LIN {X 0,Y 199.376,Z 843.056,A -85,B 0,C 180,E1 -21344.287,E2 -21344.287} C_VEL
LIN {X 0,Y 201.471,Z 836.822,A -85,B 0,C 180,E1 -21347.773,E2 -21347.773} C_VEL
LIN {X 0,Y 203.749,Z 830.038,A -85,B 0,C 180,E1 -21350.701,E2 -21350.701} C_VEL
LIN {X 0,Y 206.319,Z 821.68,A -85,B 0,C 180,E1 -21353.542,E2 -21353.542} C_VEL
LIN {X 0,Y 208.991,Z 812.769,A -85,B 0,C 180,E1 -21355.925,E2 -21355.925} C_VEL
LIN {X 0,Y 212.11,Z 801.995,A -85,B 0,C 180,E1 -21358.176,E2 -21358.176} C_VEL
LIN {X 0,Y 214.813,Z 791.098,A -85,B 0,C 180,E1 -21359.931,E2 -21359.931} C_VEL
LIN {X 0,Y 217.315,Z 778.908,A -85,B 0,C 180,E1 -21361.433,E2 -21361.433} C_VEL
LIN {X 0,Y 219.233,Z 767.366,A -85,B 0,C 180,E1 -21362.478,E2 -21362.478} C_VEL
LIN {X 0,Y 220.897,Z 754.07,A -85,B 0,C 180,E1 -21363.276,E2 -21363.276} C_VEL
LIN {X 0,Y 221.812,Z 738.89,A -85,B 0,C 180,E1 -21363.832,E2 -21363.832} C_VEL
LIN {X 0,Y 223.844,Z 690.241,A -85,B 0,C 180,E1 -21365.33,E2 -21365.33} C_VEL
LIN {X 0,Y 221.912,Z 665.137,A -85,B 0,C 180,E1 -21366.665,E2 -21366.665} C_VEL
LIN {X 0,Y 218.953,Z 639.437,A -85,B 0,C 180,E1 -21368.282,E2 -21368.282} C_VEL
LIN {X 0,Y 218.22,Z 633.043,A -85,B 0,C 180,E1 -21368.759,E2 -21368.759} C_VEL
LIN {X 0,Y 218.577,Z 624.565,A -85,B 0,C 180,E1 -21370.022,E2 -21370.022} C_VEL
LIN {X 0,Y 214.349,Z 607.039,A -85,B 0,C 180,E1 -21373.836,E2 -21373.836} C_VEL
LIN {X 0,Y 212.098,Z 598.465,A -85,B 0,C 180,E1 -21375.905,E2 -21375.905} C_VEL
LIN {X 0,Y 207.217,Z 589.004,A -85,B 0,C 180,E1 -21379.24,E2 -21379.24} C_VEL
LIN {X 0,Y 203.836,Z 583.546,A -85,B 0,C 180,E1 -21381.639,E2 -21381.639} C_VEL
LIN {X 0,Y 201.926,Z 579.961,A -85,B 0,C 180,E1 -21383.181,E2 -21383.181} C_VEL
LIN {X 0,Y 200.29,Z 577.767,A -85,B 0,C 180,E1 -21384.366,E2 -21384.366} C_VEL
LIN {X 0,Y 199.63,Z 575.61,A -85,B 0,C 180,E1 -21385.255,E2 -21385.255} C_VEL
LIN {X 0,Y 199.697,Z 575.587,A -85,B 0,C 180,E1 -21388.136,E2 -21388.136} C_VEL
LIN {X 0,Y 199.69,Z 575.605,A -85,B 0,C 180,E1 -21392.772,E2 -21392.772} C_VEL
LIN {X 0,Y 199.718,Z 575.592,A -85,B 0,C 180,E1 -21397.227,E2 -21397.227} C_VEL
LIN {X 0,Y 199.799,Z 575.564,A -85,B 0,C 180,E1 -21401.759,E2 -21401.759} C_VEL
LIN {X 0,Y 199.837,Z 575.594,A -85,B 0,C 180,E1 -21405.748,E2 -21405.748} C_VEL
LIN {X 0,Y 200.026,Z 575.533,A -85,B 0,C 180,E1 -21409.882,E2 -21409.882} C_VEL
LIN {X 0,Y 200.026,Z 575.568,A -85,B 0,C 180,E1 -21413.949,E2 -21413.949} C_VEL
LIN {X 0,Y 200.323,Z 575.496,A -85,B 0,C 180,E1 -21417.99,E2 -21417.99} C_VEL
LIN {X 0,Y 200.479,Z 575.502,A -85,B 0,C 180,E1 -21420,E2 -21420} C_VEL
LIN {X 0,Y 200.03,Z 575.536,A -85,B 0,C 180,E1 -21424.03,E2 -21424.03} C_VEL
LIN {X 0,Y 200.114,Z 575.554,A -85,B 0,C 180,E1 -21428.076,E2 -21428.076} C_VEL
LIN {X 0,Y 200.04,Z 575.55,A -85,B 0,C 180,E1 -21430.347,E2 -21430.347} C_VEL
LIN {X 0,Y 199.808,Z 575.596,A -85,B 0,C 180,E1 -21436.343,E2 -21436.343} C_VEL
LIN {X 0,Y 199.704,Z 575.587,A -85,B 0,C 180,E1 -21440.605,E2 -21440.605} C_VEL
LIN {X 0,Y 199.676,Z 575.589,A -85,B 0,C 180,E1 -21444.984,E2 -21444.984} C_VEL
LIN {X 0,Y 199.66,Z 575.671,A -85,B 0,C 180,E1 -21449.597,E2 -21449.597} C_VEL
LIN {X 0,Y 200.238,Z 577.621,A -85,B 0,C 180,E1 -21450.592,E2 -21450.592} C_VEL
LIN {X 0,Y 201.666,Z 580.137,A -85,B 0,C 180,E1 -21452.107,E2 -21452.107} C_VEL
LIN {X 0,Y 204.816,Z 586.849,A -85,B 0,C 180,E1 -21455.686,E2 -21455.686} C_VEL
LIN {X 0,Y 208.857,Z 596.996,A -85,B 0,C 180,E1 -21460.373,E2 -21460.373} C_VEL
LIN {X 0,Y 212.009,Z 606.282,A -85,B 0,C 180,E1 -21464.119,E2 -21464.119} C_VEL
LIN {X 0,Y 214.73,Z 615.526,A -85,B 0,C 180,E1 -21467.426,E2 -21467.426} C_VEL
LIN {X 0,Y 217.067,Z 625.231,A -85,B 0,C 180,E1 -21470.547,E2 -21470.547} C_VEL
LIN {X 0,Y 217.574,Z 627.419,A -85,B 0,C 180,E1 -21471.118,E2 -21471.118} C_VEL
LIN {X 0,Y 221.203,Z 635.829,A -85,B 0,C 180,E1 -21472.215,E2 -21472.215} C_VEL
LIN {X 0,Y 225.045,Z 664.563,A -85,B 0,C 180,E1 -21474.094,E2 -21474.094} C_VEL
LIN {X 0,Y 225.417,Z 668.676,A -85,B 0,C 180,E1 -21474.321,E2 -21474.321} C_VEL
LIN {X 0,Y 222.027,Z 739.582,A -85,B 0,C 180,E1 -21476.497,E2 -21476.497} C_VEL
LIN {X 0,Y 220.853,Z 752.225,A -85,B 0,C 180,E1 -21477.181,E2 -21477.181} C_VEL
LIN {X 0,Y 219.127,Z 764.44,A -85,B 0,C 180,E1 -21478.183,E2 -21478.183} C_VEL
LIN {X 0,Y 217.191,Z 775.07,A -85,B 0,C 180,E1 -21479.358,E2 -21479.358} C_VEL
LIN {X 0,Y 214.454,Z 787.114,A -85,B 0,C 180,E1 -21481.092,E2 -21481.092} C_VEL
LIN {X 0,Y 211.658,Z 797.714,A -85,B 0,C 180,E1 -21483.1,E2 -21483.1} C_VEL
LIN {X 0,Y 208.872,Z 807.539,A -85,B 0,C 180,E1 -21485.485,E2 -21485.485} C_VEL
LIN {X 0,Y 206.3,Z 815.759,A -85,B 0,C 180,E1 -21487.991,E2 -21487.991} C_VEL
LIN {X 0,Y 203.644,Z 823.224,A -85,B 0,C 180,E1 -21490.86,E2 -21490.86} C_VEL
LIN {X 0,Y 201.56,Z 829.214,A -85,B 0,C 180,E1 -21493.801,E2 -21493.801} C_VEL
LIN {X 0,Y 199.915,Z 833.946,A -85,B 0,C 180,E1 -21496.789,E2 -21496.789} C_VEL
LIN {X 0,Y 198.731,Z 837.559,A -85,B 0,C 180,E1 -21499.814,E2 -21499.814} C_VEL
LIN {X 0,Y 198.161,Z 839.419,A -85,B 0,C 180,E1 -21501.843,E2 -21501.843} C_VEL
LIN {X 0,Y 197.641,Z 841.261,A -85,B 0,C 180,E1 -21504.667,E2 -21504.667} C_VEL
LIN {X 0,Y 197.397,Z 842.439,A -85,B 0,C 180,E1 -21507.958,E2 -21507.958} C_VEL
LIN {X 0,Y 197.399,Z 842.669,A -85,B 0,C 180,E1 -21509.998,E2 -21509.998} C_VEL
LIN {X 0,Y 197.379,Z 842.473,A -85,B 0,C 180,E1 -21512.039,E2 -21512.039} C_VEL
LIN {X 0,Y 197.765,Z 840.915,A -85,B 0,C 180,E1 -21516.118,E2 -21516.118} C_VEL
LIN {X 0,Y 198.157,Z 839.543,A -85,B 0,C 180,E1 -21518.154,E2 -21518.154} C_VEL
LIN {X 0,Y 199.041,Z 836.661,A -85,B 0,C 180,E1 -21521.196,E2 -21521.196} C_VEL
LIN {X 0,Y 200.358,Z 832.739,A -85,B 0,C 180,E1 -21524.212,E2 -21524.212} C_VEL
LIN {X 0,Y 202.134,Z 827.658,A -85,B 0,C 180,E1 -21527.188,E2 -21527.188} C_VEL
LIN {X 0,Y 204.412,Z 821.25,A -85,B 0,C 180,E1 -21530.107,E2 -21530.107} C_VEL
LIN {X 0,Y 207.218,Z 813.27,A -85,B 0,C 180,E1 -21532.954,E2 -21532.954} C_VEL
LIN {X 0,Y 209.758,Z 804.815,A -85,B 0,C 180,E1 -21535.376,E2 -21535.376} C_VEL
LIN {X 0,Y 212.511,Z 795.054,A -85,B 0,C 180,E1 -21537.578,E2 -21537.578} C_VEL
LIN {X 0,Y 215.082,Z 785.125,A -85,B 0,C 180,E1 -21539.347,E2 -21539.347} C_VEL
LIN {X 0,Y 217.429,Z 774.318,A -85,B 0,C 180,E1 -21540.87,E2 -21540.87} C_VEL
LIN {X 0,Y 219.557,Z 762.357,A -85,B 0,C 180,E1 -21542.149,E2 -21542.149} C_VEL
LIN {X 0,Y 221.179,Z 749.901,A -85,B 0,C 180,E1 -21543.1,E2 -21543.1} C_VEL
LIN {X 0,Y 222.278,Z 737.222,A -85,B 0,C 180,E1 -21543.728,E2 -21543.728} C_VEL
LIN {X 0,Y 225.333,Z 671.392,A -85,B 0,C 180,E1 -21545.738,E2 -21545.738} C_VEL
LIN {X 0,Y 223.232,Z 655.911,A -85,B 0,C 180,E1 -21546.737,E2 -21546.737} C_VEL
LIN {X 0,Y 219.777,Z 634.786,A -85,B 0,C 180,E1 -21548.273,E2 -21548.273} C_VEL
LIN {X 0,Y 216.645,Z 627.6,A -85,B 0,C 180,E1 -21549.285,E2 -21549.285} C_VEL
LIN {X 0,Y 215.672,Z 627.608,A -85,B 0,C 180,E1 -21549.503,E2 -21549.503} C_VEL
LIN {X 0,Y 214.082,Z 629.763,A -85,B 0,C 180,E1 -21549.702,E2 -21549.702} C_VEL
LIN {X 0,Y 212.932,Z 631.087,A -85,B 0,C 180,E1 -21549.903,E2 -21549.903} C_VEL
LIN {X 0,Y 211.461,Z 631.109,A -85,B 0,C 180,E1 -21550.237,E2 -21550.237} C_VEL
LIN {X 0,Y 210.574,Z 629.639,A -85,B 0,C 180,E1 -21550.506,E2 -21550.506} C_VEL
LIN {X 0,Y 210.223,Z 628.001,A -85,B 0,C 180,E1 -21550.671,E2 -21550.671} C_VEL
LIN {X 0,Y 209.975,Z 627.554,A -85,B 0,C 180,E1 -21550.868,E2 -21550.868} C_VEL
LIN {X 0,Y 209.013,Z 661.135,A -85,B 0,C 180,E1 -21552.558,E2 -21552.558} C_VEL
LIN {X 0,Y 208.249,Z 675.161,A -85,B 0,C 180,E1 -21553.658,E2 -21553.658} C_VEL
LIN {X 0,Y 207.163,Z 689.066,A -85,B 0,C 180,E1 -21555.193,E2 -21555.193} C_VEL
LIN {X 0,Y 205.976,Z 701.306,A -85,B 0,C 180,E1 -21556.967,E2 -21556.967} C_VEL
LIN {X 0,Y 204.576,Z 713.727,A -85,B 0,C 180,E1 -21559.252,E2 -21559.252} C_VEL
LIN {X 0,Y 203.312,Z 723.628,A -85,B 0,C 180,E1 -21561.521,E2 -21561.521} C_VEL
LIN {X 0,Y 202.091,Z 733.699,A -85,B 0,C 180,E1 -21564.373,E2 -21564.373} C_VEL
LIN {X 0,Y 201.177,Z 741.175,A -85,B 0,C 180,E1 -21566.97,E2 -21566.97} C_VEL
LIN {X 0,Y 200.519,Z 748.385,A -85,B 0,C 180,E1 -21570.036,E2 -21570.036} C_VEL
LIN {X 0,Y 200.122,Z 753.722,A -85,B 0,C 180,E1 -21572.836,E2 -21572.836} C_VEL
LIN {X 0,Y 200.06,Z 758.466,A -85,B 0,C 180,E1 -21575.969,E2 -21575.969} C_VEL
LIN {X 0,Y 200.524,Z 762.436,A -85,B 0,C 180,E1 -21579.483,E2 -21579.483} C_VEL
LIN {X 0,Y 201.076,Z 764.264,A -85,B 0,C 180,E1 -21581.665,E2 -21581.665} C_VEL
LIN {X 0,Y 201.845,Z 765.542,A -85,B 0,C 180,E1 -21583.826,E2 -21583.826} C_VEL
LIN {X 0,Y 202.818,Z 766.369,A -85,B 0,C 180,E1 -21585.978,E2 -21585.978} C_VEL
LIN {X 0,Y 204.018,Z 766.722,A -85,B 0,C 180,E1 -21588.072,E2 -21588.072} C_VEL
LIN {X 0,Y 206.228,Z 766.345,A -85,B 0,C 180,E1 -21591.204,E2 -21591.204} C_VEL
LIN {X 0,Y 208.844,Z 764.942,A -85,B 0,C 180,E1 -21594.206,E2 -21594.206} C_VEL
LIN {X 0,Y 211.219,Z 763.1,A -85,B 0,C 180,E1 -21596.524,E2 -21596.524} C_VEL
LIN {X 0,Y 214.247,Z 760.206,A -85,B 0,C 180,E1 -21599.06,E2 -21599.06} C_VEL
LIN {X 0,Y 218.012,Z 755.835,A -85,B 0,C 180,E1 -21601.847,E2 -21601.847} C_VEL
LIN {X 0,Y 222.275,Z 750.161,A -85,B 0,C 180,E1 -21604.534,E2 -21604.534} C_VEL
LIN {X 0,Y 226.866,Z 742.967,A -85,B 0,C 180,E1 -21607.118,E2 -21607.118} C_VEL
LIN {X 0,Y 231.669,Z 734.065,A -85,B 0,C 180,E1 -21609.605,E2 -21609.605} C_VEL
LIN {X 0,Y 236.461,Z 723.753,A -85,B 0,C 180,E1 -21611.791,E2 -21611.791} C_VEL
LIN {X 0,Y 240.467,Z 713.449,A -85,B 0,C 180,E1 -21613.522,E2 -21613.522} C_VEL
LIN {X 0,Y 244.029,Z 701.968,A -85,B 0,C 180,E1 -21615.038,E2 -21615.038} C_VEL
LIN {X 0,Y 245.05,Z 696.962,A -85,B 0,C 180,E1 -21615.739,E2 -21615.739} C_VEL
LIN {X 0,Y 245.616,Z 689.046,A -85,B 0,C 180,E1 -21617.134,E2 -21617.134} C_VEL
LIN {X 0,Y 245.924,Z 680.855,A -85,B 0,C 180,E1 -21618.409,E2 -21618.409} C_VEL
LIN {X 0,Y 246.461,Z 675.44,A -85,B 0,C 180,E1 -21618.918,E2 -21618.918} C_VEL
LIN {X 0,Y 249.571,Z 650.857,A -85,B 0,C 180,E1 -21620.206,E2 -21620.206} C_VEL
LIN {X 0,Y 250.153,Z 646.426,A -85,B 0,C 180,E1 -21620.424,E2 -21620.424} C_VEL
LIN {X 0,Y 248.082,Z 641.857,A -85,B 0,C 180,E1 -21622.351,E2 -21622.351} C_VEL
LIN {X 0,Y 246.401,Z 638.478,A -85,B 0,C 180,E1 -21624.264,E2 -21624.264} C_VEL
LIN {X 0,Y 244.337,Z 636.415,A -85,B 0,C 180,E1 -21626.921,E2 -21626.921} C_VEL
LIN {X 0,Y 242.313,Z 636.359,A -85,B 0,C 180,E1 -21631.471,E2 -21631.471} C_VEL
LIN {X 0,Y 242.029,Z 637.453,A -85,B 0,C 180,E1 -21633.593,E2 -21633.593} C_VEL
LIN {X 0,Y 242.252,Z 640.017,A -85,B 0,C 180,E1 -21636.149,E2 -21636.149} C_VEL
LIN {X 0,Y 243.693,Z 646.744,A -85,B 0,C 180,E1 -21640.038,E2 -21640.038} C_VEL
LIN {X 0,Y 244.457,Z 650.053,A -85,B 0,C 180,E1 -21641.394,E2 -21641.394} C_VEL
LIN {X 0,Y 245.563,Z 654.466,A -85,B 0,C 180,E1 -21642.967,E2 -21642.967} C_VEL
LIN {X 0,Y 246.515,Z 658.782,A -85,B 0,C 180,E1 -21644.224,E2 -21644.224} C_VEL
LIN {X 0,Y 245.896,Z 673.924,A -85,B 0,C 180,E1 -21645.758,E2 -21645.758} C_VEL
LIN {X 0,Y 244.774,Z 689.882,A -85,B 0,C 180,E1 -21646.984,E2 -21646.984} C_VEL
LIN {X 0,Y 244.081,Z 696.611,A -85,B 0,C 180,E1 -21647.382,E2 -21647.382} C_VEL
LIN {X 0,Y 241.31,Z 711.484,A -85,B 0,C 180,E1 -21648.087,E2 -21648.087} C_VEL
LIN {X 0,Y 237.61,Z 725.575,A -85,B 0,C 180,E1 -21648.987,E2 -21648.987} C_VEL
LIN {X 0,Y 233.041,Z 739.08,A -85,B 0,C 180,E1 -21650.147,E2 -21650.147} C_VEL
LIN {X 0,Y 227.776,Z 751.778,A -85,B 0,C 180,E1 -21651.617,E2 -21651.617} C_VEL
LIN {X 0,Y 222.272,Z 763.259,A -85,B 0,C 180,E1 -21653.361,E2 -21653.361} C_VEL
LIN {X 0,Y 216.595,Z 773.724,A -85,B 0,C 180,E1 -21655.403,E2 -21655.403} C_VEL
LIN {X 0,Y 210.95,Z 783.143,A -85,B 0,C 180,E1 -21657.79,E2 -21657.79} C_VEL
LIN {X 0,Y 210.163,Z 784.755,A -85,B 0,C 180,E1 -21658.22,E2 -21658.22} C_VEL
LIN {X 0,Y 207.263,Z 796.997,A -85,B 0,C 180,E1 -21659.992,E2 -21659.992} C_VEL
LIN {X 0,Y 204.247,Z 807.724,A -85,B 0,C 180,E1 -21662.044,E2 -21662.044} C_VEL
LIN {X 0,Y 200.959,Z 818.25,A -85,B 0,C 180,E1 -21664.636,E2 -21664.636} C_VEL
LIN {X 0,Y 198.092,Z 827.068,A -85,B 0,C 180,E1 -21667.467,E2 -21667.467} C_VEL
LIN {X 0,Y 195.445,Z 834.658,A -85,B 0,C 180,E1 -21670.574,E2 -21670.574} C_VEL
LIN {X 0,Y 193.663,Z 839.604,A -85,B 0,C 180,E1 -21673.125,E2 -21673.125} C_VEL
LIN {X 0,Y 192.069,Z 844.394,A -85,B 0,C 180,E1 -21676.243,E2 -21676.243} C_VEL
LIN {X 0,Y 191.044,Z 848.058,A -85,B 0,C 180,E1 -21679.403,E2 -21679.403} C_VEL
LIN {X 0,Y 190.578,Z 849.948,A -85,B 0,C 180,E1 -21681.519,E2 -21681.519} C_VEL
LIN {X 0,Y 190.321,Z 851.372,A -85,B 0,C 180,E1 -21683.642,E2 -21683.642} C_VEL
LIN {X 0,Y 190.238,Z 852.44,A -85,B 0,C 180,E1 -21685.921,E2 -21685.921} C_VEL
LIN {X 0,Y 190.381,Z 853.216,A -85,B 0,C 180,E1 -21690.002,E2 -21690.002} C_VEL
LIN {X 0,Y 190.235,Z 852.424,A -85,B 0,C 180,E1 -21694.064,E2 -21694.064} C_VEL
LIN {X 0,Y 190.324,Z 851.34,A -85,B 0,C 180,E1 -21696.362,E2 -21696.362} C_VEL
LIN {X 0,Y 190.582,Z 849.898,A -85,B 0,C 180,E1 -21698.484,E2 -21698.484} C_VEL
LIN {X 0,Y 191.316,Z 846.911,A -85,B 0,C 180,E1 -21701.658,E2 -21701.658} C_VEL
LIN {X 0,Y 192.463,Z 842.862,A -85,B 0,C 180,E1 -21704.811,E2 -21704.811} C_VEL
LIN {X 0,Y 194.701,Z 836.629,A -85,B 0,C 180,E1 -21708.413,E2 -21708.413} C_VEL
LIN {X 0,Y 197.054,Z 829.98,A -85,B 0,C 180,E1 -21711.379,E2 -21711.379} C_VEL
LIN {X 0,Y 199.351,Z 822.889,A -85,B 0,C 180,E1 -21713.919,E2 -21713.919} C_VEL
LIN {X 0,Y 202.025,Z 814.508,A -85,B 0,C 180,E1 -21716.332,E2 -21716.332} C_VEL
LIN {X 0,Y 205.192,Z 804.136,A -85,B 0,C 180,E1 -21718.655,E2 -21718.655} C_VEL
LIN {X 0,Y 208.344,Z 792.457,A -85,B 0,C 180,E1 -21720.679,E2 -21720.679} C_VEL
LIN {X 0,Y 210.886,Z 780.679,A -85,B 0,C 180,E1 -21722.224,E2 -21722.224} C_VEL
LIN {X 0,Y 213.068,Z 768.472,A -85,B 0,C 180,E1 -21723.398,E2 -21723.398} C_VEL
LIN {X 0,Y 214.843,Z 755.964,A -85,B 0,C 180,E1 -21724.209,E2 -21724.209} C_VEL
LIN {X 0,Y 215.781,Z 742.593,A -85,B 0,C 180,E1 -21724.761,E2 -21724.761} C_VEL
LIN {X 0,Y 218.04,Z 690.784,A -85,B 0,C 180,E1 -21726.393,E2 -21726.393} C_VEL
LIN {X 0,Y 216.288,Z 666.684,A -85,B 0,C 180,E1 -21727.715,E2 -21727.715} C_VEL
LIN {X 0,Y 213.485,Z 641.41,A -85,B 0,C 180,E1 -21729.362,E2 -21729.362} C_VEL
LIN {X 0,Y 212.474,Z 633.523,A -85,B 0,C 180,E1 -21729.924,E2 -21729.924} C_VEL
LIN {X 0,Y 212.772,Z 627.098,A -85,B 0,C 180,E1 -21730.924,E2 -21730.924} C_VEL
LIN {X 0,Y 208.979,Z 610.361,A -85,B 0,C 180,E1 -21734.729,E2 -21734.729} C_VEL
LIN {X 0,Y 206.944,Z 602.434,A -85,B 0,C 180,E1 -21736.722,E2 -21736.722} C_VEL
LIN {X 0,Y 202.859,Z 594.437,A -85,B 0,C 180,E1 -21739.659,E2 -21739.659} C_VEL
LIN {X 0,Y 199.698,Z 589.173,A -85,B 0,C 180,E1 -21741.984,E2 -21741.984} C_VEL
LIN {X 0,Y 197.193,Z 584.939,A -85,B 0,C 180,E1 -21743.98,E2 -21743.98} C_VEL
LIN {X 0,Y 194.973,Z 580.965,A -85,B 0,C 180,E1 -21746.004,E2 -21746.004} C_VEL
LIN {X 0,Y 193.382,Z 578.923,A -85,B 0,C 180,E1 -21747.4,E2 -21747.4} C_VEL
LIN {X 0,Y 192.624,Z 576.465,A -85,B 0,C 180,E1 -21748.52,E2 -21748.52} C_VEL
LIN {X 0,Y 192.668,Z 576.484,A -85,B 0,C 180,E1 -21751.692,E2 -21751.692} C_VEL
LIN {X 0,Y 192.688,Z 576.457,A -85,B 0,C 180,E1 -21756.346,E2 -21756.346} C_VEL
LIN {X 0,Y 192.734,Z 576.445,A -85,B 0,C 180,E1 -21761.459,E2 -21761.459} C_VEL
LIN {X 0,Y 192.765,Z 576.471,A -85,B 0,C 180,E1 -21765.214,E2 -21765.214} C_VEL
LIN {X 0,Y 192.949,Z 576.413,A -85,B 0,C 180,E1 -21769.567,E2 -21769.567} C_VEL
LIN {X 0,Y 192.988,Z 576.446,A -85,B 0,C 180,E1 -21773.728,E2 -21773.728} C_VEL
LIN {X 0,Y 193.265,Z 576.374,A -85,B 0,C 180,E1 -21777.916,E2 -21777.916} C_VEL
LIN {X 0,Y 193.443,Z 576.377,A -85,B 0,C 180,E1 -21780,E2 -21780} C_VEL
LIN {X 0,Y 192.977,Z 576.412,A -85,B 0,C 180,E1 -21784.177,E2 -21784.177} C_VEL
LIN {X 0,Y 193.065,Z 576.435,A -85,B 0,C 180,E1 -21788.373,E2 -21788.373} C_VEL
LIN {X 0,Y 192.813,Z 576.434,A -85,B 0,C 180,E1 -21792.633,E2 -21792.633} C_VEL
LIN {X 0,Y 192.761,Z 576.463,A -85,B 0,C 180,E1 -21796.959,E2 -21796.959} C_VEL
LIN {X 0,Y 192.641,Z 576.476,A -85,B 0,C 180,E1 -21801.397,E2 -21801.397} C_VEL
LIN {X 0,Y 192.668,Z 576.465,A -85,B 0,C 180,E1 -21804.224,E2 -21804.224} C_VEL
LIN {X 0,Y 192.615,Z 576.495,A -85,B 0,C 180,E1 -21806.404,E2 -21806.404} C_VEL
LIN {X 0,Y 193.635,Z 579.261,A -85,B 0,C 180,E1 -21808.154,E2 -21808.154} C_VEL
LIN {X 0,Y 194.623,Z 580.578,A -85,B 0,C 180,E1 -21809.2,E2 -21809.2} C_VEL
LIN {X 0,Y 195.237,Z 582.498,A -85,B 0,C 180,E1 -21810.263,E2 -21810.263} C_VEL
LIN {X 0,Y 196.603,Z 585.04,A -85,B 0,C 180,E1 -21811.821,E2 -21811.821} C_VEL
LIN {X 0,Y 200.155,Z 593.08,A -85,B 0,C 180,E1 -21816.137,E2 -21816.137} C_VEL
LIN {X 0,Y 203.735,Z 602.268,A -85,B 0,C 180,E1 -21820.419,E2 -21820.419} C_VEL
LIN {X 0,Y 207.029,Z 612.418,A -85,B 0,C 180,E1 -21824.528,E2 -21824.528} C_VEL
LIN {X 0,Y 209.571,Z 621.855,A -85,B 0,C 180,E1 -21827.877,E2 -21827.877} C_VEL
LIN {X 0,Y 210.949,Z 627.51,A -85,B 0,C 180,E1 -21829.65,E2 -21829.65} C_VEL
LIN {X 0,Y 215.698,Z 638.078,A -85,B 0,C 180,E1 -21831.163,E2 -21831.163} C_VEL
LIN {X 0,Y 219.195,Z 664.408,A -85,B 0,C 180,E1 -21832.968,E2 -21832.968} C_VEL
LIN {X 0,Y 219.676,Z 668.777,A -85,B 0,C 180,E1 -21833.239,E2 -21833.239} C_VEL
LIN {X 0,Y 216.148,Z 739.712,A -85,B 0,C 180,E1 -21835.459,E2 -21835.459} C_VEL
LIN {X 0,Y 214.938,Z 752.387,A -85,B 0,C 180,E1 -21836.158,E2 -21836.158} C_VEL
LIN {X 0,Y 213.145,Z 764.613,A -85,B 0,C 180,E1 -21837.179,E2 -21837.179} C_VEL
LIN {X 0,Y 211.108,Z 775.251,A -85,B 0,C 180,E1 -21838.375,E2 -21838.375} C_VEL
LIN {X 0,Y 208.272,Z 787.299,A -85,B 0,C 180,E1 -21840.149,E2 -21840.149} C_VEL
LIN {X 0,Y 205.36,Z 797.902,A -85,B 0,C 180,E1 -21842.205,E2 -21842.205} C_VEL
LIN {X 0,Y 202.639,Z 807.109,A -85,B 0,C 180,E1 -21844.482,E2 -21844.482} C_VEL
LIN {X 0,Y 199.725,Z 815.95,A -85,B 0,C 180,E1 -21847.226,E2 -21847.226} C_VEL
LIN {X 0,Y 196.942,Z 823.417,A -85,B 0,C 180,E1 -21850.182,E2 -21850.182} C_VEL
LIN {X 0,Y 194.749,Z 829.407,A -85,B 0,C 180,E1 -21853.218,E2 -21853.218} C_VEL
LIN {X 0,Y 192.991,Z 834.14,A -85,B 0,C 180,E1 -21856.306,E2 -21856.306} C_VEL
LIN {X 0,Y 191.741,Z 837.753,A -85,B 0,C 180,E1 -21859.438,E2 -21859.438} C_VEL
LIN {X 0,Y 191.124,Z 839.613,A -85,B 0,C 180,E1 -21861.54,E2 -21861.54} C_VEL
LIN {X 0,Y 190.529,Z 841.647,A -85,B 0,C 180,E1 -21864.839,E2 -21864.839} C_VEL
LIN {X 0,Y 190.306,Z 842.632,A -85,B 0,C 180,E1 -21867.882,E2 -21867.882} C_VEL
LIN {X 0,Y 190.303,Z 842.862,A -85,B 0,C 180,E1 -21869.998,E2 -21869.998} C_VEL
LIN {X 0,Y 190.29,Z 842.666,A -85,B 0,C 180,E1 -21872.115,E2 -21872.115} C_VEL
LIN {X 0,Y 190.721,Z 841.107,A -85,B 0,C 180,E1 -21876.345,E2 -21876.345} C_VEL
LIN {X 0,Y 191.12,Z 839.735,A -85,B 0,C 180,E1 -21878.456,E2 -21878.456} C_VEL
LIN {X 0,Y 192.084,Z 836.852,A -85,B 0,C 180,E1 -21881.607,E2 -21881.607} C_VEL
LIN {X 0,Y 193.464,Z 832.93,A -85,B 0,C 180,E1 -21884.73,E2 -21884.73} C_VEL
LIN {X 0,Y 195.336,Z 827.848,A -85,B 0,C 180,E1 -21887.806,E2 -21887.806} C_VEL
LIN {X 0,Y 197.761,Z 821.438,A -85,B 0,C 180,E1 -21890.814,E2 -21890.814} C_VEL
LIN {X 0,Y 200.692,Z 813.456,A -85,B 0,C 180,E1 -21893.746,E2 -21893.746} C_VEL
LIN {X 0,Y 203.263,Z 805.306,A -85,B 0,C 180,E1 -21896.151,E2 -21896.151} C_VEL
LIN {X 0,Y 206.247,Z 795.234,A -85,B 0,C 180,E1 -21898.491,E2 -21898.491} C_VEL
LIN {X 0,Y 208.94,Z 785.3,A -85,B 0,C 180,E1 -21900.299,E2 -21900.299} C_VEL
LIN {X 0,Y 211.386,Z 774.487,A -85,B 0,C 180,E1 -21901.855,E2 -21901.855} C_VEL
LIN {X 0,Y 213.59,Z 762.513,A -85,B 0,C 180,E1 -21903.161,E2 -21903.161} C_VEL
LIN {X 0,Y 215.276,Z 750.037,A -85,B 0,C 180,E1 -21904.13,E2 -21904.13} C_VEL
LIN {X 0,Y 216.426,Z 737.317,A -85,B 0,C 180,E1 -21904.769,E2 -21904.769} C_VEL
LIN {X 0,Y 219.537,Z 671.342,A -85,B 0,C 180,E1 -21906.839,E2 -21906.839} C_VEL
LIN {X 0,Y 215.312,Z 642.421,A -85,B 0,C 180,E1 -21908.896,E2 -21908.896} C_VEL
LIN {X 0,Y 214.472,Z 637.87,A -85,B 0,C 180,E1 -21909.27,E2 -21909.27} C_VEL
LIN {X 0,Y 212.744,Z 638.292,A -85,B 0,C 180,E1 -21909.634,E2 -21909.634} C_VEL
LIN {X 0,Y 209.799,Z 647.838,A -85,B 0,C 180,E1 -21909.885,E2 -21909.885} C_VEL
LIN {X 0,Y 207.148,Z 653.742,A -85,B 0,C 180,E1 -21910.238,E2 -21910.238} C_VEL
LIN {X 0,Y 205.314,Z 655.78,A -85,B 0,C 180,E1 -21910.58,E2 -21910.58} C_VEL
LIN {X 0,Y 203.954,Z 655.757,A -85,B 0,C 180,E1 -21910.91,E2 -21910.91} C_VEL
LIN {X 0,Y 203.054,Z 654.326,A -85,B 0,C 180,E1 -21911.197,E2 -21911.197} C_VEL
LIN {X 0,Y 202.428,Z 651.03,A -85,B 0,C 180,E1 -21911.506,E2 -21911.506} C_VEL
LIN {X 0,Y 201.892,Z 666.8,A -85,B 0,C 180,E1 -21912.484,E2 -21912.484} C_VEL
LIN {X 0,Y 201.012,Z 680.159,A -85,B 0,C 180,E1 -21913.694,E2 -21913.694} C_VEL
LIN {X 0,Y 199.898,Z 693.275,A -85,B 0,C 180,E1 -21915.319,E2 -21915.319} C_VEL
LIN {X 0,Y 198.511,Z 706.128,A -85,B 0,C 180,E1 -21917.383,E2 -21917.383} C_VEL
LIN {X 0,Y 197.12,Z 717.644,A -85,B 0,C 180,E1 -21919.743,E2 -21919.743} C_VEL
LIN {X 0,Y 195.774,Z 728.106,A -85,B 0,C 180,E1 -21922.39,E2 -21922.39} C_VEL
LIN {X 0,Y 194.631,Z 737,A -85,B 0,C 180,E1 -21925.178,E2 -21925.178} C_VEL
LIN {X 0,Y 193.774,Z 745.052,A -85,B 0,C 180,E1 -21928.271,E2 -21928.271} C_VEL
LIN {X 0,Y 193.187,Z 752.348,A -85,B 0,C 180,E1 -21931.775,E2 -21931.775} C_VEL
LIN {X 0,Y 192.961,Z 758.438,A -85,B 0,C 180,E1 -21935.575,E2 -21935.575} C_VEL
LIN {X 0,Y 193.292,Z 762.19,A -85,B 0,C 180,E1 -21938.679,E2 -21938.679} C_VEL
LIN {X 0,Y 193.78,Z 764.339,A -85,B 0,C 180,E1 -21940.949,E2 -21940.949} C_VEL
LIN {X 0,Y 194.512,Z 765.944,A -85,B 0,C 180,E1 -21943.199,E2 -21943.199} C_VEL
LIN {X 0,Y 195.684,Z 767.254,A -85,B 0,C 180,E1 -21945.851,E2 -21945.851} C_VEL
LIN {X 0,Y 198.042,Z 767.906,A -85,B 0,C 180,E1 -21949.779,E2 -21949.779} C_VEL
LIN {X 0,Y 199.647,Z 767.652,A -85,B 0,C 180,E1 -21951.905,E2 -21951.905} C_VEL
LIN {X 0,Y 201.477,Z 766.903,A -85,B 0,C 180,E1 -21953.993,E2 -21953.993} C_VEL
LIN {X 0,Y 204.161,Z 765.284,A -85,B 0,C 180,E1 -21956.606,E2 -21956.606} C_VEL
LIN {X 0,Y 208.235,Z 761.815,A -85,B 0,C 180,E1 -21960,E2 -21960} C_VEL
LIN {X 0,Y 212.677,Z 757.152,A -85,B 0,C 180,E1 -21963.111,E2 -21963.111} C_VEL
LIN {X 0,Y 216.77,Z 752.092,A -85,B 0,C 180,E1 -21965.582,E2 -21965.582} C_VEL
LIN {X 0,Y 221.604,Z 745.092,A -85,B 0,C 180,E1 -21968.205,E2 -21968.205} C_VEL
LIN {X 0,Y 226.7,Z 736.465,A -85,B 0,C 180,E1 -21970.72,E2 -21970.72} C_VEL
LIN {X 0,Y 231.028,Z 728.02,A -85,B 0,C 180,E1 -21972.621,E2 -21972.621} C_VEL
LIN {X 0,Y 235.47,Z 717.633,A -85,B 0,C 180,E1 -21974.475,E2 -21974.475} C_VEL
LIN {X 0,Y 239.259,Z 707.117,A -85,B 0,C 180,E1 -21975.985,E2 -21975.985} C_VEL
LIN {X 0,Y 242.677,Z 695.266,A -85,B 0,C 180,E1 -21977.311,E2 -21977.311} C_VEL
LIN {X 0,Y 245.529,Z 681.532,A -85,B 0,C 180,E1 -21978.5,E2 -21978.5} C_VEL
LIN {X 0,Y 246.461,Z 675.44,A -85,B 0,C 180,E1 -21978.918,E2 -21978.918} C_VEL
LIN {X 0,Y 246.683,Z 671.773,A -85,B 0,C 180,E1 -21979.289,E2 -21979.289} C_VEL
LIN {X 0,Y 245.909,Z 660.831,A -85,B 0,C 180,E1 -21981.125,E2 -21981.125} C_VEL
LIN {X 0,Y 246.184,Z 657.118,A -85,B 0,C 180,E1 -21981.444,E2 -21981.444} C_VEL
LIN {X 0,Y 247.061,Z 650.673,A -85,B 0,C 180,E1 -21981.768,E2 -21981.768} C_VEL
LIN {X 0,Y 245.213,Z 646.558,A -85,B 0,C 180,E1 -21983.826,E2 -21983.826} C_VEL
LIN {X 0,Y 244.331,Z 644.872,A -85,B 0,C 180,E1 -21984.901,E2 -21984.901} C_VEL
LIN {X 0,Y 242.843,Z 643.398,A -85,B 0,C 180,E1 -21986.988,E2 -21986.988} C_VEL
LIN {X 0,Y 241.402,Z 643.193,A -85,B 0,C 180,E1 -21989.665,E2 -21989.665} C_VEL
LIN {X 0,Y 240.788,Z 643.55,A -85,B 0,C 180,E1 -21992.178,E2 -21992.178} C_VEL
LIN {X 0,Y 240.703,Z 645.949,A -85,B 0,C 180,E1 -21995.165,E2 -21995.165} C_VEL
LIN {X 0,Y 241.3,Z 650.878,A -85,B 0,C 180,E1 -21998.221,E2 -21998.221} C_VEL
LIN {X 0,Y 242.177,Z 654.865,A -85,B 0,C 180,E1 -22000.2,E2 -22000.2} C_VEL
LIN {X 0,Y 243.188,Z 660.085,A -85,B 0,C 180,E1 -22002.11,E2 -22002.11} C_VEL
LIN {X 0,Y 243.796,Z 663.303,A -85,B 0,C 180,E1 -22003.034,E2 -22003.034} C_VEL
LIN {X 0,Y 242.794,Z 678.616,A -85,B 0,C 180,E1 -22004.547,E2 -22004.547} C_VEL
LIN {X 0,Y 241.477,Z 693.803,A -85,B 0,C 180,E1 -22005.696,E2 -22005.696} C_VEL
LIN {X 0,Y 239.035,Z 707.689,A -85,B 0,C 180,E1 -22006.369,E2 -22006.369} C_VEL
LIN {X 0,Y 235.308,Z 721.81,A -85,B 0,C 180,E1 -22007.2,E2 -22007.2} C_VEL
LIN {X 0,Y 230.875,Z 734.764,A -85,B 0,C 180,E1 -22008.252,E2 -22008.252} C_VEL
LIN {X 0,Y 225.335,Z 748.072,A -85,B 0,C 180,E1 -22009.674,E2 -22009.674} C_VEL
LIN {X 0,Y 219.444,Z 759.98,A -85,B 0,C 180,E1 -22011.356,E2 -22011.356} C_VEL
LIN {X 0,Y 213.974,Z 769.811,A -85,B 0,C 180,E1 -22013.174,E2 -22013.174} C_VEL
LIN {X 0,Y 207.839,Z 779.616,A -85,B 0,C 180,E1 -22015.503,E2 -22015.503} C_VEL
LIN {X 0,Y 203.888,Z 785.888,A -85,B 0,C 180,E1 -22017.341,E2 -22017.341} C_VEL
LIN {X 0,Y 201.143,Z 796.821,A -85,B 0,C 180,E1 -22018.98,E2 -22018.98} C_VEL
LIN {X 0,Y 197.978,Z 807.542,A -85,B 0,C 180,E1 -22021.077,E2 -22021.077} C_VEL
LIN {X 0,Y 194.542,Z 818.064,A -85,B 0,C 180,E1 -22023.736,E2 -22023.736} C_VEL
LIN {X 0,Y 191.722,Z 826.257,A -85,B 0,C 180,E1 -22026.41,E2 -22026.41} C_VEL
LIN {X 0,Y 189.112,Z 833.355,A -85,B 0,C 180,E1 -22029.328,E2 -22029.328} C_VEL
LIN {X 0,Y 186.85,Z 839.413,A -85,B 0,C 180,E1 -22032.49,E2 -22032.49} C_VEL
LIN {X 0,Y 185.139,Z 844.202,A -85,B 0,C 180,E1 -22035.717,E2 -22035.717} C_VEL
LIN {X 0,Y 184.049,Z 847.866,A -85,B 0,C 180,E1 -22038.995,E2 -22038.995} C_VEL
LIN {X 0,Y 183.541,Z 849.755,A -85,B 0,C 180,E1 -22041.192,E2 -22041.192} C_VEL
LIN {X 0,Y 183.243,Z 851.179,A -85,B 0,C 180,E1 -22043.395,E2 -22043.395} C_VEL
LIN {X 0,Y 183.129,Z 852.41,A -85,B 0,C 180,E1 -22046.208,E2 -22046.208} C_VEL
LIN {X 0,Y 183.281,Z 853.023,A -85,B 0,C 180,E1 -22050.002,E2 -22050.002} C_VEL
LIN {X 0,Y 183.15,Z 852.353,A -85,B 0,C 180,E1 -22053.889,E2 -22053.889} C_VEL
LIN {X 0,Y 183.246,Z 851.146,A -85,B 0,C 180,E1 -22056.609,E2 -22056.609} C_VEL
LIN {X 0,Y 183.544,Z 849.704,A -85,B 0,C 180,E1 -22058.812,E2 -22058.812} C_VEL
LIN {X 0,Y 184.342,Z 846.717,A -85,B 0,C 180,E1 -22062.106,E2 -22062.106} C_VEL
LIN {X 0,Y 185.57,Z 842.668,A -85,B 0,C 180,E1 -22065.375,E2 -22065.375} C_VEL
LIN {X 0,Y 187.952,Z 836.436,A -85,B 0,C 180,E1 -22069.1,E2 -22069.1} C_VEL
LIN {X 0,Y 190.603,Z 829.279,A -85,B 0,C 180,E1 -22072.376,E2 -22072.376} C_VEL
LIN {X 0,Y 193.339,Z 821.135,A -85,B 0,C 180,E1 -22075.286,E2 -22075.286} C_VEL
LIN {X 0,Y 196.295,Z 812.391,A -85,B 0,C 180,E1 -22077.74,E2 -22077.74} C_VEL
LIN {X 0,Y 199.695,Z 801.623,A -85,B 0,C 180,E1 -22080.101,E2 -22080.101} C_VEL
LIN {X 0,Y 202.616,Z 790.732,A -85,B 0,C 180,E1 -22081.937,E2 -22081.937} C_VEL
LIN {X 0,Y 205.295,Z 778.552,A -85,B 0,C 180,E1 -22083.507,E2 -22083.507} C_VEL
LIN {X 0,Y 207.41,Z 767.031,A -85,B 0,C 180,E1 -22084.582,E2 -22084.582} C_VEL
LIN {X 0,Y 209.162,Z 754.156,A -85,B 0,C 180,E1 -22085.387,E2 -22085.387} C_VEL
LIN {X 0,Y 210.188,Z 738.65,A -85,B 0,C 180,E1 -22085.985,E2 -22085.985} C_VEL
LIN {X 0,Y 212.375,Z 692.028,A -85,B 0,C 180,E1 -22087.472,E2 -22087.472} C_VEL
LIN {X 0,Y 210.524,Z 666.234,A -85,B 0,C 180,E1 -22088.953,E2 -22088.953} C_VEL
LIN {X 0,Y 207.896,Z 641.626,A -85,B 0,C 180,E1 -22090.623,E2 -22090.623} C_VEL
LIN {X 0,Y 206.918,Z 632.695,A -85,B 0,C 180,E1 -22091.337,E2 -22091.337} C_VEL
LIN {X 0,Y 207.118,Z 630.284,A -85,B 0,C 180,E1 -22091.711,E2 -22091.711} C_VEL
LIN {X 0,Y 203.759,Z 614.309,A -85,B 0,C 180,E1 -22095.497,E2 -22095.497} C_VEL
LIN {X 0,Y 202.11,Z 607.333,A -85,B 0,C 180,E1 -22097.305,E2 -22097.305} C_VEL
LIN {X 0,Y 199.139,Z 601.205,A -85,B 0,C 180,E1 -22099.54,E2 -22099.54} C_VEL
LIN {X 0,Y 194.89,Z 593.773,A -85,B 0,C 180,E1 -22102.841,E2 -22102.841} C_VEL
LIN {X 0,Y 193.106,Z 590.575,A -85,B 0,C 180,E1 -22104.387,E2 -22104.387} C_VEL
LIN {X 0,Y 190.914,Z 586.574,A -85,B 0,C 180,E1 -22106.483,E2 -22106.483} C_VEL
LIN {X 0,Y 189.16,Z 584.197,A -85,B 0,C 180,E1 -22108.032,E2 -22108.032} C_VEL
LIN {X 0,Y 188.191,Z 582.002,A -85,B 0,C 180,E1 -22109.199,E2 -22109.199} C_VEL
LIN {X 0,Y 186.58,Z 580.168,A -85,B 0,C 180,E1 -22110.681,E2 -22110.681} C_VEL
LIN {X 0,Y 185.571,Z 577.368,A -85,B 0,C 180,E1 -22112.359,E2 -22112.359} C_VEL
LIN {X 0,Y 185.584,Z 577.337,A -85,B 0,C 180,E1 -22115.382,E2 -22115.382} C_VEL
LIN {X 0,Y 185.677,Z 577.325,A -85,B 0,C 180,E1 -22121.135,E2 -22121.135} C_VEL
LIN {X 0,Y 185.697,Z 577.339,A -85,B 0,C 180,E1 -22124.637,E2 -22124.637} C_VEL
LIN {X 0,Y 185.892,Z 577.292,A -85,B 0,C 180,E1 -22129.418,E2 -22129.418} C_VEL
LIN {X 0,Y 185.951,Z 577.324,A -85,B 0,C 180,E1 -22133.49,E2 -22133.49} C_VEL
LIN {X 0,Y 186.209,Z 577.252,A -85,B 0,C 180,E1 -22137.837,E2 -22137.837} C_VEL
LIN {X 0,Y 186.407,Z 577.252,A -85,B 0,C 180,E1 -22140,E2 -22140} C_VEL
LIN {X 0,Y 185.924,Z 577.289,A -85,B 0,C 180,E1 -22144.336,E2 -22144.336} C_VEL
LIN {X 0,Y 186.012,Z 577.315,A -85,B 0,C 180,E1 -22148.693,E2 -22148.693} C_VEL
LIN {X 0,Y 185.737,Z 577.316,A -85,B 0,C 180,E1 -22153.122,E2 -22153.122} C_VEL
LIN {X 0,Y 185.694,Z 577.333,A -85,B 0,C 180,E1 -22157.625,E2 -22157.625} C_VEL
LIN {X 0,Y 185.601,Z 577.366,A -85,B 0,C 180,E1 -22162.691,E2 -22162.691} C_VEL
LIN {X 0,Y 186.487,Z 579.995,A -85,B 0,C 180,E1 -22164.491,E2 -22164.491} C_VEL
LIN {X 0,Y 187.906,Z 581.89,A -85,B 0,C 180,E1 -22166.149,E2 -22166.149} C_VEL
LIN {X 0,Y 188.818,Z 584.264,A -85,B 0,C 180,E1 -22167.727,E2 -22167.727} C_VEL
LIN {X 0,Y 189.733,Z 585.601,A -85,B 0,C 180,E1 -22168.786,E2 -22168.786} C_VEL
LIN {X 0,Y 192.877,Z 592.879,A -85,B 0,C 180,E1 -22173.132,E2 -22173.132} C_VEL
LIN {X 0,Y 195.91,Z 600.203,A -85,B 0,C 180,E1 -22177.049,E2 -22177.049} C_VEL
LIN {X 0,Y 199.082,Z 608.878,A -85,B 0,C 180,E1 -22181.034,E2 -22181.034} C_VEL
LIN {X 0,Y 202.307,Z 619.659,A -85,B 0,C 180,E1 -22185.315,E2 -22185.315} C_VEL
LIN {X 0,Y 204.343,Z 627.646,A -85,B 0,C 180,E1 -22188.059,E2 -22188.059} C_VEL
LIN {X 0,Y 210.064,Z 640.232,A -85,B 0,C 180,E1 -22190.005,E2 -22190.005} C_VEL
LIN {X 0,Y 210.716,Z 642.758,A -85,B 0,C 180,E1 -22190.264,E2 -22190.264} C_VEL
LIN {X 0,Y 213.983,Z 669.295,A -85,B 0,C 180,E1 -22192.109,E2 -22192.109} C_VEL
LIN {X 0,Y 210.346,Z 739.845,A -85,B 0,C 180,E1 -22194.364,E2 -22194.364} C_VEL
LIN {X 0,Y 209.092,Z 752.549,A -85,B 0,C 180,E1 -22195.077,E2 -22195.077} C_VEL
LIN {X 0,Y 207.233,Z 764.787,A -85,B 0,C 180,E1 -22196.119,E2 -22196.119} C_VEL
LIN {X 0,Y 205.089,Z 775.431,A -85,B 0,C 180,E1 -22197.334,E2 -22197.334} C_VEL
LIN {X 0,Y 202.145,Z 787.484,A -85,B 0,C 180,E1 -22199.147,E2 -22199.147} C_VEL
LIN {X 0,Y 199.111,Z 798.09,A -85,B 0,C 180,E1 -22201.253,E2 -22201.253} C_VEL
LIN {X 0,Y 196.114,Z 807.713,A -85,B 0,C 180,E1 -22203.705,E2 -22203.705} C_VEL
LIN {X 0,Y 193.191,Z 816.142,A -85,B 0,C 180,E1 -22206.41,E2 -22206.41} C_VEL
LIN {X 0,Y 190.28,Z 823.609,A -85,B 0,C 180,E1 -22209.457,E2 -22209.457} C_VEL
LIN {X 0,Y 187.941,Z 829.6,A -85,B 0,C 180,E1 -22212.591,E2 -22212.591} C_VEL
LIN {X 0,Y 186.083,Z 834.333,A -85,B 0,C 180,E1 -22215.787,E2 -22215.787} C_VEL
LIN {X 0,Y 184.753,Z 837.947,A -85,B 0,C 180,E1 -22219.034,E2 -22219.034} C_VEL
LIN {X 0,Y 184.114,Z 839.806,A -85,B 0,C 180,E1 -22221.216,E2 -22221.216} C_VEL
LIN {X 0,Y 183.397,Z 842.039,A -85,B 0,C 180,E1 -22225.107,E2 -22225.107} C_VEL
LIN {X 0,Y 183.217,Z 842.825,A -85,B 0,C 180,E1 -22227.8,E2 -22227.8} C_VEL
LIN {X 0,Y 183.209,Z 843.055,A -85,B 0,C 180,E1 -22229.998,E2 -22229.998} C_VEL
LIN {X 0,Y 183.202,Z 842.859,A -85,B 0,C 180,E1 -22232.197,E2 -22232.197} C_VEL
LIN {X 0,Y 183.682,Z 841.299,A -85,B 0,C 180,E1 -22236.589,E2 -22236.589} C_VEL
LIN {X 0,Y 184.11,Z 839.927,A -85,B 0,C 180,E1 -22238.781,E2 -22238.781} C_VEL
LIN {X 0,Y 185.116,Z 837.044,A -85,B 0,C 180,E1 -22242.051,E2 -22242.051} C_VEL
LIN {X 0,Y 186.587,Z 833.121,A -85,B 0,C 180,E1 -22245.285,E2 -22245.285} C_VEL
LIN {X 0,Y 188.573,Z 828.038,A -85,B 0,C 180,E1 -22248.467,E2 -22248.467} C_VEL
LIN {X 0,Y 191.138,Z 821.626,A -85,B 0,C 180,E1 -22251.571,E2 -22251.571} C_VEL
LIN {X 0,Y 194.19,Z 813.643,A -85,B 0,C 180,E1 -22254.593,E2 -22254.593} C_VEL
LIN {X 0,Y 197.135,Z 804.764,A -85,B 0,C 180,E1 -22257.26,E2 -22257.26} C_VEL
LIN {X 0,Y 200.371,Z 794.273,A -85,B 0,C 180,E1 -22259.696,E2 -22259.696} C_VEL
LIN {X 0,Y 203.227,Z 784.093,A -85,B 0,C 180,E1 -22261.535,E2 -22261.535} C_VEL
LIN {X 0,Y 205.776,Z 772.908,A -85,B 0,C 180,E1 -22263.122,E2 -22263.122} C_VEL
LIN {X 0,Y 208.075,Z 760.202,A -85,B 0,C 180,E1 -22264.452,E2 -22264.452} C_VEL
LIN {X 0,Y 209.798,Z 747.619,A -85,B 0,C 180,E1 -22265.371,E2 -22265.371} C_VEL
LIN {X 0,Y 210.867,Z 734.376,A -85,B 0,C 180,E1 -22265.972,E2 -22265.972} C_VEL
LIN {X 0,Y 213.875,Z 672.44,A -85,B 0,C 180,E1 -22267.94,E2 -22267.94} C_VEL
LIN {X 0,Y 211.791,Z 657.036,A -85,B 0,C 180,E1 -22269.04,E2 -22269.04} C_VEL
LIN {X 0,Y 208.772,Z 660.898,A -85,B 0,C 180,E1 -22269.546,E2 -22269.546} C_VEL
LIN {X 0,Y 206.107,Z 662.627,A -85,B 0,C 180,E1 -22270.084,E2 -22270.084} C_VEL
LIN {X 0,Y 205.078,Z 662.918,A -85,B 0,C 180,E1 -22270.314,E2 -22270.314} C_VEL
LIN {X 0,Y 201.995,Z 670.722,A -85,B 0,C 180,E1 -22270.701,E2 -22270.701} C_VEL
LIN {X 0,Y 199.455,Z 674.865,A -85,B 0,C 180,E1 -22271.138,E2 -22271.138} C_VEL
LIN {X 0,Y 197.529,Z 676.793,A -85,B 0,C 180,E1 -22271.536,E2 -22271.536} C_VEL
LIN {X 0,Y 195.856,Z 676.765,A -85,B 0,C 180,E1 -22271.973,E2 -22271.973} C_VEL
LIN {X 0,Y 194.997,Z 675.328,A -85,B 0,C 180,E1 -22272.272,E2 -22272.272} C_VEL
LIN {X 0,Y 194.6,Z 672.914,A -85,B 0,C 180,E1 -22272.527,E2 -22272.527} C_VEL
LIN {X 0,Y 193.569,Z 686.638,A -85,B 0,C 180,E1 -22273.999,E2 -22273.999} C_VEL
LIN {X 0,Y 192.41,Z 698.516,A -85,B 0,C 180,E1 -22275.688,E2 -22275.688} C_VEL
LIN {X 0,Y 190.912,Z 711.301,A -85,B 0,C 180,E1 -22277.995,E2 -22277.995} C_VEL
LIN {X 0,Y 189.501,Z 722.536,A -85,B 0,C 180,E1 -22280.571,E2 -22280.571} C_VEL
LIN {X 0,Y 188.208,Z 732.254,A -85,B 0,C 180,E1 -22283.311,E2 -22283.311} C_VEL
LIN {X 0,Y 187.126,Z 741.041,A -85,B 0,C 180,E1 -22286.36,E2 -22286.36} C_VEL
LIN {X 0,Y 186.482,Z 747.911,A -85,B 0,C 180,E1 -22289.279,E2 -22289.279} C_VEL
LIN {X 0,Y 185.938,Z 754.985,A -85,B 0,C 180,E1 -22293.027,E2 -22293.027} C_VEL
LIN {X 0,Y 185.969,Z 760.265,A -85,B 0,C 180,E1 -22296.621,E2 -22296.621} C_VEL
LIN {X 0,Y 186.55,Z 764.347,A -85,B 0,C 180,E1 -22300.355,E2 -22300.355} C_VEL
LIN {X 0,Y 187.168,Z 766.133,A -85,B 0,C 180,E1 -22302.519,E2 -22302.519} C_VEL
LIN {X 0,Y 188.53,Z 768.017,A -85,B 0,C 180,E1 -22305.738,E2 -22305.738} C_VEL
LIN {X 0,Y 190.64,Z 769.054,A -85,B 0,C 180,E1 -22309.378,E2 -22309.378} C_VEL
LIN {X 0,Y 192.273,Z 769.103,A -85,B 0,C 180,E1 -22311.593,E2 -22311.593} C_VEL
LIN {X 0,Y 194.079,Z 768.66,A -85,B 0,C 180,E1 -22313.763,E2 -22313.763} C_VEL
LIN {X 0,Y 197.093,Z 767.265,A -85,B 0,C 180,E1 -22316.744,E2 -22316.744} C_VEL
LIN {X 0,Y 200.971,Z 764.588,A -85,B 0,C 180,E1 -22320,E2 -22320} C_VEL
LIN {X 0,Y 204.599,Z 761.391,A -85,B 0,C 180,E1 -22322.626,E2 -22322.626} C_VEL
LIN {X 0,Y 209.684,Z 755.999,A -85,B 0,C 180,E1 -22325.771,E2 -22325.771} C_VEL
LIN {X 0,Y 214.77,Z 749.73,A -85,B 0,C 180,E1 -22328.468,E2 -22328.468} C_VEL
LIN {X 0,Y 220.025,Z 741.902,A -85,B 0,C 180,E1 -22331.049,E2 -22331.049} C_VEL
LIN {X 0,Y 225.129,Z 733.091,A -85,B 0,C 180,E1 -22333.292,E2 -22333.292} C_VEL
LIN {X 0,Y 230.094,Z 723.041,A -85,B 0,C 180,E1 -22335.274,E2 -22335.274} C_VEL
LIN {X 0,Y 234.596,Z 712.016,A -85,B 0,C 180,E1 -22336.983,E2 -22336.983} C_VEL
LIN {X 0,Y 238.427,Z 700.121,A -85,B 0,C 180,E1 -22338.423,E2 -22338.423} C_VEL
LIN {X 0,Y 241.419,Z 688.45,A -85,B 0,C 180,E1 -22339.53,E2 -22339.53} C_VEL
LIN {X 0,Y 243.741,Z 675.406,A -85,B 0,C 180,E1 -22340.483,E2 -22340.483} C_VEL
LIN {X 0,Y 246.184,Z 657.118,A -85,B 0,C 180,E1 -22341.444,E2 -22341.444} C_VEL
LIN {X 0,Y 246.248,Z 655.045,A -85,B 0,C 180,E1 -22341.702,E2 -22341.702} C_VEL
LIN {X 0,Y 245.823,Z 653.247,A -85,B 0,C 180,E1 -22342.278,E2 -22342.278} C_VEL
LIN {X 0,Y 244.775,Z 652.004,A -85,B 0,C 180,E1 -22343.279,E2 -22343.279} C_VEL
LIN {X 0,Y 242.502,Z 651.455,A -85,B 0,C 180,E1 -22345.414,E2 -22345.414} C_VEL
LIN {X 0,Y 241.943,Z 651.029,A -85,B 0,C 180,E1 -22346.132,E2 -22346.132} C_VEL
LIN {X 0,Y 241.256,Z 650.314,A -85,B 0,C 180,E1 -22347.18,E2 -22347.18} C_VEL
LIN {X 0,Y 239.879,Z 650.166,A -85,B 0,C 180,E1 -22349.872,E2 -22349.872} C_VEL
LIN {X 0,Y 239.306,Z 650.717,A -85,B 0,C 180,E1 -22352.401,E2 -22352.401} C_VEL
LIN {X 0,Y 239.202,Z 653.224,A -85,B 0,C 180,E1 -22355.134,E2 -22355.134} C_VEL
LIN {X 0,Y 239.926,Z 659.302,A -85,B 0,C 180,E1 -22358.733,E2 -22358.733} C_VEL
LIN {X 0,Y 240.872,Z 664.688,A -85,B 0,C 180,E1 -22360.91,E2 -22360.91} C_VEL
LIN {X 0,Y 241.213,Z 667.579,A -85,B 0,C 180,E1 -22361.765,E2 -22361.765} C_VEL
LIN {X 0,Y 240.077,Z 681.543,A -85,B 0,C 180,E1 -22363.139,E2 -22363.139} C_VEL
LIN {X 0,Y 238.476,Z 696.469,A -85,B 0,C 180,E1 -22364.258,E2 -22364.258} C_VEL
LIN {X 0,Y 235.295,Z 711.018,A -85,B 0,C 180,E1 -22364.97,E2 -22364.97} C_VEL
LIN {X 0,Y 230.965,Z 725.279,A -85,B 0,C 180,E1 -22365.891,E2 -22365.891} C_VEL
LIN {X 0,Y 225.722,Z 738.826,A -85,B 0,C 180,E1 -22367.074,E2 -22367.074} C_VEL
LIN {X 0,Y 220.058,Z 751.005,A -85,B 0,C 180,E1 -22368.497,E2 -22368.497} C_VEL
LIN {X 0,Y 214.015,Z 762.019,A -85,B 0,C 180,E1 -22370.184,E2 -22370.184} C_VEL
LIN {X 0,Y 207.297,Z 772.977,A -85,B 0,C 180,E1 -22372.395,E2 -22372.395} C_VEL
LIN {X 0,Y 201.102,Z 781.997,A -85,B 0,C 180,E1 -22374.789,E2 -22374.789} C_VEL
LIN {X 0,Y 197.646,Z 787.012,A -85,B 0,C 180,E1 -22376.404,E2 -22376.404} C_VEL
LIN {X 0,Y 194.712,Z 797.935,A -85,B 0,C 180,E1 -22378.14,E2 -22378.14} C_VEL
LIN {X 0,Y 191.446,Z 808.418,A -85,B 0,C 180,E1 -22380.294,E2 -22380.294} C_VEL
LIN {X 0,Y 188.169,Z 817.879,A -85,B 0,C 180,E1 -22382.775,E2 -22382.775} C_VEL
LIN {X 0,Y 184.936,Z 826.75,A -85,B 0,C 180,E1 -22385.791,E2 -22385.791} C_VEL
LIN {X 0,Y 182.474,Z 833.167,A -85,B 0,C 180,E1 -22388.54,E2 -22388.54} C_VEL
LIN {X 0,Y 180.07,Z 839.222,A -85,B 0,C 180,E1 -22391.808,E2 -22391.808} C_VEL
LIN {X 0,Y 178.234,Z 844.01,A -85,B 0,C 180,E1 -22395.151,E2 -22395.151} C_VEL
LIN {X 0,Y 177.044,Z 847.673,A -85,B 0,C 180,E1 -22398.554,E2 -22398.554} C_VEL
LIN {X 0,Y 176.497,Z 849.562,A -85,B 0,C 180,E1 -22400.837,E2 -22400.837} C_VEL
LIN {X 0,Y 176.164,Z 850.986,A -85,B 0,C 180,E1 -22403.128,E2 -22403.128} C_VEL
LIN {X 0,Y 176.03,Z 852.351,A -85,B 0,C 180,E1 -22406.495,E2 -22406.495} C_VEL
LIN {X 0,Y 176.184,Z 852.829,A -85,B 0,C 180,E1 -22410.002,E2 -22410.002} C_VEL
LIN {X 0,Y 176.06,Z 852.292,A -85,B 0,C 180,E1 -22413.665,E2 -22413.665} C_VEL
LIN {X 0,Y 176.166,Z 850.952,A -85,B 0,C 180,E1 -22416.876,E2 -22416.876} C_VEL
LIN {X 0,Y 176.501,Z 849.51,A -85,B 0,C 180,E1 -22419.167,E2 -22419.167} C_VEL
LIN {X 0,Y 177.39,Z 846.523,A -85,B 0,C 180,E1 -22422.588,E2 -22422.588} C_VEL
LIN {X 0,Y 178.701,Z 842.474,A -85,B 0,C 180,E1 -22425.981,E2 -22425.981} C_VEL
LIN {X 0,Y 181.209,Z 836.242,A -85,B 0,C 180,E1 -22429.84,E2 -22429.84} C_VEL
LIN {X 0,Y 183.919,Z 829.368,A -85,B 0,C 180,E1 -22433.099,E2 -22433.099} C_VEL
LIN {X 0,Y 186.925,Z 820.944,A -85,B 0,C 180,E1 -22436.219,E2 -22436.219} C_VEL
LIN {X 0,Y 190.032,Z 812.201,A -85,B 0,C 180,E1 -22438.738,E2 -22438.738} C_VEL
LIN {X 0,Y 193.554,Z 801.435,A -85,B 0,C 180,E1 -22441.161,E2 -22441.161} C_VEL
LIN {X 0,Y 196.615,Z 790.549,A -85,B 0,C 180,E1 -22443.034,E2 -22443.034} C_VEL
LIN {X 0,Y 199.426,Z 778.376,A -85,B 0,C 180,E1 -22444.631,E2 -22444.631} C_VEL
LIN {X 0,Y 201.619,Z 766.864,A -85,B 0,C 180,E1 -22445.725,E2 -22445.725} C_VEL
LIN {X 0,Y 203.396,Z 754.191,A -85,B 0,C 180,E1 -22446.536,E2 -22446.536} C_VEL
LIN {X 0,Y 204.451,Z 739.274,A -85,B 0,C 180,E1 -22447.129,E2 -22447.129} C_VEL
LIN {X 0,Y 206.709,Z 692.493,A -85,B 0,C 180,E1 -22448.661,E2 -22448.661} C_VEL
LIN {X 0,Y 205.026,Z 667.188,A -85,B 0,C 180,E1 -22450.16,E2 -22450.16} C_VEL
LIN {X 0,Y 202.421,Z 642.055,A -85,B 0,C 180,E1 -22451.942,E2 -22451.942} C_VEL
LIN {X 0,Y 201.38,Z 633.158,A -85,B 0,C 180,E1 -22452.642,E2 -22452.642} C_VEL
LIN {X 0,Y 199.382,Z 622.638,A -85,B 0,C 180,E1 -22455.172,E2 -22455.172} C_VEL
LIN {X 0,Y 197.057,Z 611.415,A -85,B 0,C 180,E1 -22458.152,E2 -22458.152} C_VEL
LIN {X 0,Y 193.86,Z 604.944,A -85,B 0,C 180,E1 -22460.623,E2 -22460.623} C_VEL
LIN {X 0,Y 189.455,Z 596.893,A -85,B 0,C 180,E1 -22464.381,E2 -22464.381} C_VEL
LIN {X 0,Y 186.797,Z 592.174,A -85,B 0,C 180,E1 -22466.938,E2 -22466.938} C_VEL
LIN {X 0,Y 185.019,Z 589.633,A -85,B 0,C 180,E1 -22468.612,E2 -22468.612} C_VEL
LIN {X 0,Y 184.508,Z 588.279,A -85,B 0,C 180,E1 -22469.308,E2 -22469.308} C_VEL
LIN {X 0,Y 182.597,Z 585.742,A -85,B 0,C 180,E1 -22471.242,E2 -22471.242} C_VEL
LIN {X 0,Y 181.44,Z 583.125,A -85,B 0,C 180,E1 -22472.988,E2 -22472.988} C_VEL
LIN {X 0,Y 179.56,Z 581.075,A -85,B 0,C 180,E1 -22475.28,E2 -22475.28} C_VEL
LIN {X 0,Y 178.526,Z 578.233,A -85,B 0,C 180,E1 -22477.582,E2 -22477.582} C_VEL
LIN {X 0,Y 178.652,Z 578.197,A -85,B 0,C 180,E1 -22481.657,E2 -22481.657} C_VEL
LIN {X 0,Y 178.66,Z 578.227,A -85,B 0,C 180,E1 -22486.348,E2 -22486.348} C_VEL
LIN {X 0,Y 178.915,Z 578.166,A -85,B 0,C 180,E1 -22490.96,E2 -22490.96} C_VEL
LIN {X 0,Y 178.868,Z 578.177,A -85,B 0,C 180,E1 -22495.493,E2 -22495.493} C_VEL
LIN {X 0,Y 179.371,Z 578.126,A -85,B 0,C 180,E1 -22500,E2 -22500} C_VEL
LIN {X 0,Y 178.872,Z 578.166,A -85,B 0,C 180,E1 -22504.507,E2 -22504.507} C_VEL
LIN {X 0,Y 178.963,Z 578.193,A -85,B 0,C 180,E1 -22509.038,E2 -22509.038} C_VEL
LIN {X 0,Y 178.67,Z 578.199,A -85,B 0,C 180,E1 -22513.651,E2 -22513.651} C_VEL
LIN {X 0,Y 178.669,Z 578.283,A -85,B 0,C 180,E1 -22517.897,E2 -22517.897} C_VEL
LIN {X 0,Y 179.765,Z 581.396,A -85,B 0,C 180,E1 -22520.601,E2 -22520.601} C_VEL
LIN {X 0,Y 181.23,Z 583.465,A -85,B 0,C 180,E1 -22522.818,E2 -22522.818} C_VEL
LIN {X 0,Y 184.878,Z 590.643,A -85,B 0,C 180,E1 -22528.372,E2 -22528.372} C_VEL
LIN {X 0,Y 187.609,Z 597.187,A -85,B 0,C 180,E1 -22532.454,E2 -22532.454} C_VEL
LIN {X 0,Y 190.399,Z 603.959,A -85,B 0,C 180,E1 -22536.199,E2 -22536.199} C_VEL
LIN {X 0,Y 193.76,Z 613.554,A -85,B 0,C 180,E1 -22540.76,E2 -22540.76} C_VEL
LIN {X 0,Y 196.672,Z 623.652,A -85,B 0,C 180,E1 -22544.863,E2 -22544.863} C_VEL
LIN {X 0,Y 197.749,Z 627.786,A -85,B 0,C 180,E1 -22546.319,E2 -22546.319} C_VEL
LIN {X 0,Y 203.259,Z 639.43,A -85,B 0,C 180,E1 -22548.333,E2 -22548.333} C_VEL
LIN {X 0,Y 205.285,Z 644.195,A -85,B 0,C 180,E1 -22549.053,E2 -22549.053} C_VEL
LIN {X 0,Y 208.414,Z 670.698,A -85,B 0,C 180,E1 -22550.965,E2 -22550.965} C_VEL
LIN {X 0,Y 204.635,Z 739.977,A -85,B 0,C 180,E1 -22553.209,E2 -22553.209} C_VEL
LIN {X 0,Y 203.332,Z 752.71,A -85,B 0,C 180,E1 -22553.936,E2 -22553.936} C_VEL
LIN {X 0,Y 201.566,Z 763.883,A -85,B 0,C 180,E1 -22554.878,E2 -22554.878} C_VEL
LIN {X 0,Y 199.162,Z 775.612,A -85,B 0,C 180,E1 -22556.234,E2 -22556.234} C_VEL
LIN {X 0,Y 196.098,Z 787.669,A -85,B 0,C 180,E1 -22558.086,E2 -22558.086} C_VEL
LIN {X 0,Y 192.929,Z 798.277,A -85,B 0,C 180,E1 -22560.241,E2 -22560.241} C_VEL
LIN {X 0,Y 189.829,Z 807.694,A -85,B 0,C 180,E1 -22562.692,E2 -22562.692} C_VEL
LIN {X 0,Y 186.7,Z 816.333,A -85,B 0,C 180,E1 -22565.537,E2 -22565.537} C_VEL
LIN {X 0,Y 183.656,Z 823.801,A -85,B 0,C 180,E1 -22568.681,E2 -22568.681} C_VEL
LIN {X 0,Y 181.157,Z 829.794,A -85,B 0,C 180,E1 -22571.917,E2 -22571.917} C_VEL
LIN {X 0,Y 179.192,Z 834.527,A -85,B 0,C 180,E1 -22575.229,E2 -22575.229} C_VEL
LIN {X 0,Y 177.787,Z 838.14,A -85,B 0,C 180,E1 -22578.599,E2 -22578.599} C_VEL
LIN {X 0,Y 177.094,Z 840,A -85,B 0,C 180,E1 -22580.864,E2 -22580.864} C_VEL
LIN {X 0,Y 176.636,Z 841.415,A -85,B 0,C 180,E1 -22583.143,E2 -22583.143} C_VEL
LIN {X 0,Y 176.132,Z 843.018,A -85,B 0,C 180,E1 -22587.711,E2 -22587.711} C_VEL
LIN {X 0,Y 176.118,Z 843.248,A -85,B 0,C 180,E1 -22589.998,E2 -22589.998} C_VEL
LIN {X 0,Y 176.117,Z 843.051,A -85,B 0,C 180,E1 -22592.285,E2 -22592.285} C_VEL
LIN {X 0,Y 176.635,Z 841.491,A -85,B 0,C 180,E1 -22596.853,E2 -22596.853} C_VEL
LIN {X 0,Y 177.09,Z 840.119,A -85,B 0,C 180,E1 -22599.132,E2 -22599.132} C_VEL
LIN {X 0,Y 178.172,Z 837.236,A -85,B 0,C 180,E1 -22602.528,E2 -22602.528} C_VEL
LIN {X 0,Y 179.738,Z 833.312,A -85,B 0,C 180,E1 -22605.883,E2 -22605.883} C_VEL
LIN {X 0,Y 181.845,Z 828.228,A -85,B 0,C 180,E1 -22609.176,E2 -22609.176} C_VEL
LIN {X 0,Y 184.552,Z 821.815,A -85,B 0,C 180,E1 -22612.382,E2 -22612.382} C_VEL
LIN {X 0,Y 187.743,Z 813.83,A -85,B 0,C 180,E1 -22615.496,E2 -22615.496} C_VEL
LIN {X 0,Y 190.79,Z 805.101,A -85,B 0,C 180,E1 -22618.197,E2 -22618.197} C_VEL
LIN {X 0,Y 193.888,Z 795.594,A -85,B 0,C 180,E1 -22620.493,E2 -22620.493} C_VEL
LIN {X 0,Y 197.21,Z 784.268,A -85,B 0,C 180,E1 -22622.614,E2 -22622.614} C_VEL
LIN {X 0,Y 199.878,Z 773.075,A -85,B 0,C 180,E1 -22624.232,E2 -22624.232} C_VEL
LIN {X 0,Y 202.261,Z 760.355,A -85,B 0,C 180,E1 -22625.59,E2 -22625.59} C_VEL
LIN {X 0,Y 204.061,Z 747.752,A -85,B 0,C 180,E1 -22626.523,E2 -22626.523} C_VEL
LIN {X 0,Y 205.183,Z 734.446,A -85,B 0,C 180,E1 -22627.133,E2 -22627.133} C_VEL
LIN {X 0,Y 208.296,Z 673.522,A -85,B 0,C 180,E1 -22629.101,E2 -22629.101} C_VEL
LIN {X 0,Y 207.995,Z 670.838,A -85,B 0,C 180,E1 -22629.286,E2 -22629.286} C_VEL
LIN {X 0,Y 204.598,Z 677.461,A -85,B 0,C 180,E1 -22629.772,E2 -22629.772} C_VEL
LIN {X 0,Y 201.415,Z 681.49,A -85,B 0,C 180,E1 -22630.346,E2 -22630.346} C_VEL
LIN {X 0,Y 198.697,Z 683.467,A -85,B 0,C 180,E1 -22630.924,E2 -22630.924} C_VEL
LIN {X 0,Y 196.072,Z 684.137,A -85,B 0,C 180,E1 -22631.561,E2 -22631.561} C_VEL
LIN {X 0,Y 192.817,Z 689.937,A -85,B 0,C 180,E1 -22632.139,E2 -22632.139} C_VEL
LIN {X 0,Y 190.042,Z 692.914,A -85,B 0,C 180,E1 -22632.751,E2 -22632.751} C_VEL
LIN {X 0,Y 189.262,Z 693.386,A -85,B 0,C 180,E1 -22632.947,E2 -22632.947} C_VEL
LIN {X 0,Y 187.739,Z 693.416,A -85,B 0,C 180,E1 -22633.38,E2 -22633.38} C_VEL
LIN {X 0,Y 186.776,Z 692.313,A -85,B 0,C 180,E1 -22633.718,E2 -22633.718} C_VEL
LIN {X 0,Y 186.322,Z 690.039,A -85,B 0,C 180,E1 -22633.989,E2 -22633.989} C_VEL
LIN {X 0,Y 185.008,Z 702.832,A -85,B 0,C 180,E1 -22635.974,E2 -22635.974} C_VEL
LIN {X 0,Y 183.577,Z 714.578,A -85,B 0,C 180,E1 -22638.304,E2 -22638.304} C_VEL
LIN {X 0,Y 182.173,Z 724.804,A -85,B 0,C 180,E1 -22640.806,E2 -22640.806} C_VEL
LIN {X 0,Y 180.962,Z 734.343,A -85,B 0,C 180,E1 -22643.682,E2 -22643.682} C_VEL
LIN {X 0,Y 179.888,Z 742.863,A -85,B 0,C 180,E1 -22646.841,E2 -22646.841} C_VEL
LIN {X 0,Y 179.226,Z 750.141,A -85,B 0,C 180,E1 -22650.148,E2 -22650.148} C_VEL
LIN {X 0,Y 178.84,Z 755.536,A -85,B 0,C 180,E1 -22653.133,E2 -22653.133} C_VEL
LIN {X 0,Y 178.903,Z 760.962,A -85,B 0,C 180,E1 -22656.868,E2 -22656.868} C_VEL
LIN {X 0,Y 179.396,Z 764.551,A -85,B 0,C 180,E1 -22660.08,E2 -22660.08} C_VEL
LIN {X 0,Y 180.726,Z 767.887,A -85,B 0,C 180,E1 -22664.204,E2 -22664.204} C_VEL
LIN {X 0,Y 181.837,Z 769.162,A -85,B 0,C 180,E1 -22666.591,E2 -22666.591} C_VEL
LIN {X 0,Y 183.207,Z 769.991,A -85,B 0,C 180,E1 -22668.942,E2 -22668.942} C_VEL
LIN {X 0,Y 184.851,Z 770.34,A -85,B 0,C 180,E1 -22671.289,E2 -22671.289} C_VEL
LIN {X 0,Y 186.66,Z 770.217,A -85,B 0,C 180,E1 -22673.514,E2 -22673.514} C_VEL
LIN {X 0,Y 190.021,Z 769.148,A -85,B 0,C 180,E1 -22676.923,E2 -22676.923} C_VEL
LIN {X 0,Y 193.657,Z 767.138,A -85,B 0,C 180,E1 -22680,E2 -22680} C_VEL
LIN {X 0,Y 197.58,Z 764.222,A -85,B 0,C 180,E1 -22682.859,E2 -22682.859} C_VEL
LIN {X 0,Y 202.604,Z 759.701,A -85,B 0,C 180,E1 -22685.973,E2 -22685.973} C_VEL
LIN {X 0,Y 207.763,Z 754.118,A -85,B 0,C 180,E1 -22688.756,E2 -22688.756} C_VEL
LIN {X 0,Y 213.27,Z 747.017,A -85,B 0,C 180,E1 -22691.404,E2 -22691.404} C_VEL
LIN {X 0,Y 219.125,Z 738.265,A -85,B 0,C 180,E1 -22693.919,E2 -22693.919} C_VEL
LIN {X 0,Y 224.742,Z 728.137,A -85,B 0,C 180,E1 -22696.113,E2 -22696.113} C_VEL
LIN {X 0,Y 229.884,Z 717.036,A -85,B 0,C 180,E1 -22697.991,E2 -22697.991} C_VEL
LIN {X 0,Y 234.194,Z 705.536,A -85,B 0,C 180,E1 -22699.503,E2 -22699.503} C_VEL
LIN {X 0,Y 237.871,Z 692.975,A -85,B 0,C 180,E1 -22700.766,E2 -22700.766} C_VEL
LIN {X 0,Y 240.257,Z 681.604,A -85,B 0,C 180,E1 -22701.68,E2 -22701.68} C_VEL
LIN {X 0,Y 243.257,Z 661.718,A -85,B 0,C 180,E1 -22702.819,E2 -22702.819} C_VEL
LIN {X 0,Y 244.206,Z 655.211,A -85,B 0,C 180,E1 -22703.155,E2 -22703.155} C_VEL
LIN {X 0,Y 242.714,Z 651.751,A -85,B 0,C 180,E1 -22705.09,E2 -22705.09} C_VEL
LIN {X 0,Y 241.943,Z 651.029,A -85,B 0,C 180,E1 -22706.132,E2 -22706.132} C_VEL
LIN {X 0,Y 241.303,Z 650.693,A -85,B 0,C 180,E1 -22707.044,E2 -22707.044} C_VEL
LIN {X 0,Y 240.275,Z 651.467,A -85,B 0,C 180,E1 -22708.416,E2 -22708.416} C_VEL
LIN {X 0,Y 238.72,Z 654.691,A -85,B 0,C 180,E1 -22710.664,E2 -22710.664} C_VEL
LIN {X 0,Y 237.897,Z 657.552,A -85,B 0,C 180,E1 -22712.497,E2 -22712.497} C_VEL
LIN {X 0,Y 237.678,Z 658.612,A -85,B 0,C 180,E1 -22713.445,E2 -22713.445} C_VEL
LIN {X 0,Y 237.691,Z 660.357,A -85,B 0,C 180,E1 -22714.987,E2 -22714.987} C_VEL
LIN {X 0,Y 238.261,Z 666.426,A -85,B 0,C 180,E1 -22718.471,E2 -22718.471} C_VEL
LIN {X 0,Y 238.907,Z 671.624,A -85,B 0,C 180,E1 -22720.417,E2 -22720.417} C_VEL
LIN {X 0,Y 237.722,Z 683.317,A -85,B 0,C 180,E1 -22721.594,E2 -22721.594} C_VEL
LIN {X 0,Y 235.929,Z 697.475,A -85,B 0,C 180,E1 -22722.679,E2 -22722.679} C_VEL
LIN {X 0,Y 232.247,Z 712.576,A -85,B 0,C 180,E1 -22723.429,E2 -22723.429} C_VEL
LIN {X 0,Y 228.107,Z 725.136,A -85,B 0,C 180,E1 -22724.25,E2 -22724.25} C_VEL
LIN {X 0,Y 222.689,Z 738.254,A -85,B 0,C 180,E1 -22725.399,E2 -22725.399} C_VEL
LIN {X 0,Y 216.814,Z 750.189,A -85,B 0,C 180,E1 -22726.786,E2 -22726.786} C_VEL
LIN {X 0,Y 211.143,Z 760.142,A -85,B 0,C 180,E1 -22728.266,E2 -22728.266} C_VEL
LIN {X 0,Y 204.046,Z 771.104,A -85,B 0,C 180,E1 -22730.42,E2 -22730.42} C_VEL
LIN {X 0,Y 197.404,Z 780.162,A -85,B 0,C 180,E1 -22732.757,E2 -22732.757} C_VEL
LIN {X 0,Y 191.454,Z 788.029,A -85,B 0,C 180,E1 -22735.403,E2 -22735.403} C_VEL
LIN {X 0,Y 188.323,Z 799.029,A -85,B 0,C 180,E1 -22737.243,E2 -22737.243} C_VEL
LIN {X 0,Y 184.965,Z 809.293,A -85,B 0,C 180,E1 -22739.459,E2 -22739.459} C_VEL
LIN {X 0,Y 181.872,Z 817.694,A -85,B 0,C 180,E1 -22741.749,E2 -22741.749} C_VEL
LIN {X 0,Y 178.936,Z 825.436,A -85,B 0,C 180,E1 -22744.405,E2 -22744.405} C_VEL
LIN {X 0,Y 175.88,Z 832.978,A -85,B 0,C 180,E1 -22747.693,E2 -22747.693} C_VEL
LIN {X 0,Y 173.324,Z 839.032,A -85,B 0,C 180,E1 -22751.074,E2 -22751.074} C_VEL
LIN {X 0,Y 171.33,Z 843.818,A -85,B 0,C 180,E1 -22754.538,E2 -22754.538} C_VEL
LIN {X 0,Y 170.066,Z 847.481,A -85,B 0,C 180,E1 -22758.078,E2 -22758.078} C_VEL
LIN {X 0,Y 169.475,Z 849.37,A -85,B 0,C 180,E1 -22760.454,E2 -22760.454} C_VEL
LIN {X 0,Y 169.111,Z 850.793,A -85,B 0,C 180,E1 -22762.84,E2 -22762.84} C_VEL
LIN {X 0,Y 168.953,Z 852.229,A -85,B 0,C 180,E1 -22766.695,E2 -22766.695} C_VEL
LIN {X 0,Y 169.09,Z 852.637,A -85,B 0,C 180,E1 -22770.002,E2 -22770.002} C_VEL
LIN {X 0,Y 168.98,Z 852.185,A -85,B 0,C 180,E1 -22773.459,E2 -22773.459} C_VEL
LIN {X 0,Y 169.113,Z 850.759,A -85,B 0,C 180,E1 -22777.164,E2 -22777.164} C_VEL
LIN {X 0,Y 169.477,Z 849.316,A -85,B 0,C 180,E1 -22779.55,E2 -22779.55} C_VEL
LIN {X 0,Y 170.431,Z 846.329,A -85,B 0,C 180,E1 -22783.111,E2 -22783.111} C_VEL
LIN {X 0,Y 171.862,Z 842.28,A -85,B 0,C 180,E1 -22786.636,E2 -22786.636} C_VEL
LIN {X 0,Y 174.501,Z 836.048,A -85,B 0,C 180,E1 -22790.636,E2 -22790.636} C_VEL
LIN {X 0,Y 177.264,Z 829.462,A -85,B 0,C 180,E1 -22793.874,E2 -22793.874} C_VEL
LIN {X 0,Y 179.991,Z 822.314,A -85,B 0,C 180,E1 -22796.683,E2 -22796.683} C_VEL
LIN {X 0,Y 183.133,Z 813.939,A -85,B 0,C 180,E1 -22799.296,E2 -22799.296} C_VEL
LIN {X 0,Y 186.741,Z 803.574,A -85,B 0,C 180,E1 -22801.797,E2 -22801.797} C_VEL
LIN {X 0,Y 189.871,Z 793.319,A -85,B 0,C 180,E1 -22803.727,E2 -22803.727} C_VEL
LIN {X 0,Y 192.738,Z 782.072,A -85,B 0,C 180,E1 -22805.372,E2 -22805.372} C_VEL
LIN {X 0,Y 195.432,Z 769.23,A -85,B 0,C 180,E1 -22806.718,E2 -22806.718} C_VEL
LIN {X 0,Y 197.558,Z 755.906,A -85,B 0,C 180,E1 -22807.659,E2 -22807.659} C_VEL
LIN {X 0,Y 198.656,Z 742.762,A -85,B 0,C 180,E1 -22808.242,E2 -22808.242} C_VEL
LIN {X 0,Y 201.188,Z 693.216,A -85,B 0,C 180,E1 -22809.894,E2 -22809.894} C_VEL
LIN {X 0,Y 199.604,Z 668.216,A -85,B 0,C 180,E1 -22811.433,E2 -22811.433} C_VEL
LIN {X 0,Y 197.275,Z 644.435,A -85,B 0,C 180,E1 -22813.179,E2 -22813.179} C_VEL
LIN {X 0,Y 196.139,Z 635.212,A -85,B 0,C 180,E1 -22813.946,E2 -22813.946} C_VEL
LIN {X 0,Y 195.225,Z 632.46,A -85,B 0,C 180,E1 -22814.439,E2 -22814.439} C_VEL
LIN {X 0,Y 192.785,Z 619.551,A -85,B 0,C 180,E1 -22817.838,E2 -22817.838} C_VEL
LIN {X 0,Y 192.096,Z 616.065,A -85,B 0,C 180,E1 -22818.811,E2 -22818.811} C_VEL
LIN {X 0,Y 189.256,Z 609.934,A -85,B 0,C 180,E1 -22821.247,E2 -22821.247} C_VEL
LIN {X 0,Y 184.792,Z 601.709,A -85,B 0,C 180,E1 -22825.216,E2 -22825.216} C_VEL
LIN {X 0,Y 182.591,Z 597.703,A -85,B 0,C 180,E1 -22827.393,E2 -22827.393} C_VEL
LIN {X 0,Y 180.995,Z 595.336,A -85,B 0,C 180,E1 -22829.022,E2 -22829.022} C_VEL
LIN {X 0,Y 179.629,Z 592.706,A -85,B 0,C 180,E1 -22830.721,E2 -22830.721} C_VEL
LIN {X 0,Y 178.206,Z 590.317,A -85,B 0,C 180,E1 -22832.457,E2 -22832.457} C_VEL
LIN {X 0,Y 177.768,Z 589.23,A -85,B 0,C 180,E1 -22833.207,E2 -22833.207} C_VEL
LIN {X 0,Y 176.08,Z 587.439,A -85,B 0,C 180,E1 -22835.223,E2 -22835.223} C_VEL
LIN {X 0,Y 174.726,Z 584.486,A -85,B 0,C 180,E1 -22837.69,E2 -22837.69} C_VEL
LIN {X 0,Y 171.797,Z 580.196,A -85,B 0,C 180,E1 -22843.36,E2 -22843.36} C_VEL
LIN {X 0,Y 171.569,Z 579.1,A -85,B 0,C 180,E1 -22844.862,E2 -22844.862} C_VEL
LIN {X 0,Y 171.852,Z 579.042,A -85,B 0,C 180,E1 -22850.585,E2 -22850.585} C_VEL
LIN {X 0,Y 171.816,Z 579.056,A -85,B 0,C 180,E1 -22855.308,E2 -22855.308} C_VEL
LIN {X 0,Y 172.334,Z 579.001,A -85,B 0,C 180,E1 -22860,E2 -22860} C_VEL
LIN {X 0,Y 171.821,Z 579.044,A -85,B 0,C 180,E1 -22864.693,E2 -22864.693} C_VEL
LIN {X 0,Y 171.892,Z 579.067,A -85,B 0,C 180,E1 -22869.413,E2 -22869.413} C_VEL
LIN {X 0,Y 171.772,Z 579.169,A -85,B 0,C 180,E1 -22871.38,E2 -22871.38} C_VEL
LIN {X 0,Y 172.398,Z 581.577,A -85,B 0,C 180,E1 -22874.158,E2 -22874.158} C_VEL
LIN {X 0,Y 174.305,Z 583.944,A -85,B 0,C 180,E1 -22877.602,E2 -22877.602} C_VEL
LIN {X 0,Y 175.059,Z 586.278,A -85,B 0,C 180,E1 -22879.651,E2 -22879.651} C_VEL
LIN {X 0,Y 176.589,Z 588.616,A -85,B 0,C 180,E1 -22882.215,E2 -22882.215} C_VEL
LIN {X 0,Y 179.234,Z 594.278,A -85,B 0,C 180,E1 -22886.804,E2 -22886.804} C_VEL
LIN {X 0,Y 180.409,Z 596.787,A -85,B 0,C 180,E1 -22888.669,E2 -22888.669} C_VEL
LIN {X 0,Y 182.646,Z 602.208,A -85,B 0,C 180,E1 -22892.162,E2 -22892.162} C_VEL
LIN {X 0,Y 185.161,Z 608.412,A -85,B 0,C 180,E1 -22895.67,E2 -22895.67} C_VEL
LIN {X 0,Y 188.159,Z 617.271,A -85,B 0,C 180,E1 -22900.029,E2 -22900.029} C_VEL
LIN {X 0,Y 191.15,Z 627.812,A -85,B 0,C 180,E1 -22904.394,E2 -22904.394} C_VEL
LIN {X 0,Y 197.431,Z 640.691,A -85,B 0,C 180,E1 -22906.867,E2 -22906.867} C_VEL
LIN {X 0,Y 200.128,Z 647.027,A -85,B 0,C 180,E1 -22907.89,E2 -22907.89} C_VEL
LIN {X 0,Y 202.878,Z 671.094,A -85,B 0,C 180,E1 -22909.699,E2 -22909.699} C_VEL
LIN {X 0,Y 199.016,Z 740.107,A -85,B 0,C 180,E1 -22911.99,E2 -22911.99} C_VEL
LIN {X 0,Y 197.649,Z 752.872,A -85,B 0,C 180,E1 -22912.727,E2 -22912.727} C_VEL
LIN {X 0,Y 195.632,Z 765.136,A -85,B 0,C 180,E1 -22913.805,E2 -22913.805} C_VEL
LIN {X 0,Y 193.314,Z 775.792,A -85,B 0,C 180,E1 -22915.067,E2 -22915.067} C_VEL
LIN {X 0,Y 190.119,Z 787.854,A -85,B 0,C 180,E1 -22916.956,E2 -22916.956} C_VEL
LIN {X 0,Y 186.816,Z 798.465,A -85,B 0,C 180,E1 -22919.163,E2 -22919.163} C_VEL
LIN {X 0,Y 183.341,Z 808.452,A -85,B 0,C 180,E1 -22921.844,E2 -22921.844} C_VEL
LIN {X 0,Y 180.257,Z 816.525,A -85,B 0,C 180,E1 -22924.602,E2 -22924.602} C_VEL
LIN {X 0,Y 177.072,Z 823.993,A -85,B 0,C 180,E1 -22927.847,E2 -22927.847} C_VEL
LIN {X 0,Y 174.401,Z 829.987,A -85,B 0,C 180,E1 -22931.191,E2 -22931.191} C_VEL
LIN {X 0,Y 172.327,Z 834.72,A -85,B 0,C 180,E1 -22934.626,E2 -22934.626} C_VEL
LIN {X 0,Y 170.816,Z 838.334,A -85,B 0,C 180,E1 -22938.127,E2 -22938.127} C_VEL
LIN {X 0,Y 170.099,Z 840.193,A -85,B 0,C 180,E1 -22940.485,E2 -22940.485} C_VEL
LIN {X 0,Y 169.585,Z 841.608,A -85,B 0,C 180,E1 -22942.856,E2 -22942.856} C_VEL
LIN {X 0,Y 169.036,Z 843.212,A -85,B 0,C 180,E1 -22947.615,E2 -22947.615} C_VEL
LIN {X 0,Y 169.029,Z 843.44,A -85,B 0,C 180,E1 -22949.998,E2 -22949.998} C_VEL
LIN {X 0,Y 169.114,Z 842.861,A -85,B 0,C 180,E1 -22954.141,E2 -22954.141} C_VEL
LIN {X 0,Y 169.584,Z 841.684,A -85,B 0,C 180,E1 -22957.14,E2 -22957.14} C_VEL
LIN {X 0,Y 170.095,Z 840.311,A -85,B 0,C 180,E1 -22959.511,E2 -22959.511} C_VEL
LIN {X 0,Y 171.251,Z 837.427,A -85,B 0,C 180,E1 -22963.043,E2 -22963.043} C_VEL
LIN {X 0,Y 172.916,Z 833.503,A -85,B 0,C 180,E1 -22966.527,E2 -22966.527} C_VEL
LIN {X 0,Y 175.152,Z 828.417,A -85,B 0,C 180,E1 -22969.939,E2 -22969.939} C_VEL
LIN {X 0,Y 178.01,Z 822.002,A -85,B 0,C 180,E1 -22973.252,E2 -22973.252} C_VEL
LIN {X 0,Y 181.332,Z 814.017,A -85,B 0,C 180,E1 -22976.466,E2 -22976.466} C_VEL
LIN {X 0,Y 184.365,Z 805.846,A -85,B 0,C 180,E1 -22979.077,E2 -22979.077} C_VEL
LIN {X 0,Y 187.821,Z 795.773,A -85,B 0,C 180,E1 -22981.589,E2 -22981.589} C_VEL
LIN {X 0,Y 191.268,Z 784.443,A -85,B 0,C 180,E1 -22983.76,E2 -22983.76} C_VEL
LIN {X 0,Y 194.059,Z 773.241,A -85,B 0,C 180,E1 -22985.409,E2 -22985.409} C_VEL
LIN {X 0,Y 196.527,Z 760.51,A -85,B 0,C 180,E1 -22986.795,E2 -22986.795} C_VEL
LIN {X 0,Y 198.383,Z 748.085,A -85,B 0,C 180,E1 -22987.728,E2 -22987.728} C_VEL
LIN {X 0,Y 199.574,Z 734.632,A -85,B 0,C 180,E1 -22988.356,E2 -22988.356} C_VEL
LIN {X 0,Y 202.063,Z 688.881,A -85,B 0,C 180,E1 -22989.853,E2 -22989.853} C_VEL
LIN {X 0,Y 198.888,Z 690.674,A -85,B 0,C 180,E1 -22990.538,E2 -22990.538} C_VEL
LIN {X 0,Y 195.449,Z 695.847,A -85,B 0,C 180,E1 -22991.159,E2 -22991.159} C_VEL
LIN {X 0,Y 192.063,Z 699.085,A -85,B 0,C 180,E1 -22991.89,E2 -22991.89} C_VEL
LIN {X 0,Y 189.669,Z 700.305,A -85,B 0,C 180,E1 -22992.482,E2 -22992.482} C_VEL
LIN {X 0,Y 187.054,Z 700.749,A -85,B 0,C 180,E1 -22993.198,E2 -22993.198} C_VEL
LIN {X 0,Y 183.655,Z 705.438,A -85,B 0,C 180,E1 -22993.953,E2 -22993.953} C_VEL
LIN {X 0,Y 180.959,Z 707.58,A -85,B 0,C 180,E1 -22994.666,E2 -22994.666} C_VEL
LIN {X 0,Y 179.086,Z 707.699,A -85,B 0,C 180,E1 -22995.256,E2 -22995.256} C_VEL
LIN {X 0,Y 178.249,Z 706.702,A -85,B 0,C 180,E1 -22995.585,E2 -22995.585} C_VEL
LIN {X 0,Y 177.796,Z 704.708,A -85,B 0,C 180,E1 -22995.887,E2 -22995.887} C_VEL
LIN {X 0,Y 176.312,Z 716.532,A -85,B 0,C 180,E1 -22998.377,E2 -22998.377} C_VEL
LIN {X 0,Y 174.9,Z 727.012,A -85,B 0,C 180,E1 -23001.107,E2 -23001.107} C_VEL
LIN {X 0,Y 173.659,Z 736.138,A -85,B 0,C 180,E1 -23004.033,E2 -23004.033} C_VEL
LIN {X 0,Y 172.659,Z 744.644,A -85,B 0,C 180,E1 -23007.361,E2 -23007.361} C_VEL
LIN {X 0,Y 171.953,Z 752.74,A -85,B 0,C 180,E1 -23011.299,E2 -23011.299} C_VEL
LIN {X 0,Y 171.706,Z 758.766,A -85,B 0,C 180,E1 -23015.025,E2 -23015.025} C_VEL
LIN {X 0,Y 172.006,Z 763.14,A -85,B 0,C 180,E1 -23018.424,E2 -23018.424} C_VEL
LIN {X 0,Y 172.89,Z 766.92,A -85,B 0,C 180,E1 -23022.249,E2 -23022.249} C_VEL
LIN {X 0,Y 174.422,Z 769.545,A -85,B 0,C 180,E1 -23026.009,E2 -23026.009} C_VEL
LIN {X 0,Y 175.764,Z 770.709,A -85,B 0,C 180,E1 -23028.467,E2 -23028.467} C_VEL
LIN {X 0,Y 177.709,Z 771.438,A -85,B 0,C 180,E1 -23031.359,E2 -23031.359} C_VEL
LIN {X 0,Y 181.348,Z 771.352,A -85,B 0,C 180,E1 -23035.555,E2 -23035.555} C_VEL
LIN {X 0,Y 183.689,Z 770.638,A -85,B 0,C 180,E1 -23037.807,E2 -23037.807} C_VEL
LIN {X 0,Y 186.309,Z 769.467,A -85,B 0,C 180,E1 -23040,E2 -23040} C_VEL
LIN {X 0,Y 189.957,Z 767.331,A -85,B 0,C 180,E1 -23042.697,E2 -23042.697} C_VEL
LIN {X 0,Y 195.488,Z 763.129,A -85,B 0,C 180,E1 -23046.191,E2 -23046.191} C_VEL
LIN {X 0,Y 200.812,Z 758.155,A -85,B 0,C 180,E1 -23049.061,E2 -23049.061} C_VEL
LIN {X 0,Y 206.514,Z 751.843,A -85,B 0,C 180,E1 -23051.782,E2 -23051.782} C_VEL
LIN {X 0,Y 212.484,Z 743.969,A -85,B 0,C 180,E1 -23054.363,E2 -23054.363} C_VEL
LIN {X 0,Y 217.786,Z 735.886,A -85,B 0,C 180,E1 -23056.401,E2 -23056.401} C_VEL
LIN {X 0,Y 223.273,Z 726.026,A -85,B 0,C 180,E1 -23058.347,E2 -23058.347} C_VEL
LIN {X 0,Y 228.254,Z 715.182,A -85,B 0,C 180,E1 -23060.032,E2 -23060.032} C_VEL
LIN {X 0,Y 232.67,Z 703.202,A -85,B 0,C 180,E1 -23061.485,E2 -23061.485} C_VEL
LIN {X 0,Y 236.448,Z 689.912,A -85,B 0,C 180,E1 -23062.731,E2 -23062.731} C_VEL
LIN {X 0,Y 239.017,Z 676.809,A -85,B 0,C 180,E1 -23063.639,E2 -23063.639} C_VEL
LIN {X 0,Y 241.532,Z 660.064,A -85,B 0,C 180,E1 -23064.541,E2 -23064.541} C_VEL
LIN {X 0,Y 240.981,Z 658.498,A -85,B 0,C 180,E1 -23065.445,E2 -23065.445} C_VEL
LIN {X 0,Y 239.671,Z 657.233,A -85,B 0,C 180,E1 -23067.375,E2 -23067.375} C_VEL
LIN {X 0,Y 238.035,Z 657.272,A -85,B 0,C 180,E1 -23071.464,E2 -23071.464} C_VEL
LIN {X 0,Y 237.678,Z 658.612,A -85,B 0,C 180,E1 -23073.445,E2 -23073.445} C_VEL
LIN {X 0,Y 237.549,Z 660.152,A -85,B 0,C 180,E1 -23074.312,E2 -23074.312} C_VEL
LIN {X 0,Y 237.116,Z 663.598,A -85,B 0,C 180,E1 -23075.284,E2 -23075.284} C_VEL
LIN {X 0,Y 236.406,Z 670.46,A -85,B 0,C 180,E1 -23076.895,E2 -23076.895} C_VEL
LIN {X 0,Y 236.417,Z 671.982,A -85,B 0,C 180,E1 -23077.442,E2 -23077.442} C_VEL
LIN {X 0,Y 236.711,Z 676.293,A -85,B 0,C 180,E1 -23079.143,E2 -23079.143} C_VEL
LIN {X 0,Y 235.171,Z 689.093,A -85,B 0,C 180,E1 -23080.338,E2 -23080.338} C_VEL
LIN {X 0,Y 233.449,Z 699.527,A -85,B 0,C 180,E1 -23081.11,E2 -23081.11} C_VEL
LIN {X 0,Y 229.614,Z 713.454,A -85,B 0,C 180,E1 -23081.812,E2 -23081.812} C_VEL
LIN {X 0,Y 224.055,Z 728.581,A -85,B 0,C 180,E1 -23082.847,E2 -23082.847} C_VEL
LIN {X 0,Y 217.793,Z 742.131,A -85,B 0,C 180,E1 -23084.114,E2 -23084.114} C_VEL
LIN {X 0,Y 211.106,Z 754.192,A -85,B 0,C 180,E1 -23085.647,E2 -23085.647} C_VEL
LIN {X 0,Y 204.719,Z 764.114,A -85,B 0,C 180,E1 -23087.314,E2 -23087.314} C_VEL
LIN {X 0,Y 197.514,Z 774.133,A -85,B 0,C 180,E1 -23089.508,E2 -23089.508} C_VEL
LIN {X 0,Y 190.816,Z 782.43,A -85,B 0,C 180,E1 -23091.911,E2 -23091.911} C_VEL
LIN {X 0,Y 185.327,Z 789.024,A -85,B 0,C 180,E1 -23094.337,E2 -23094.337} C_VEL
LIN {X 0,Y 181.982,Z 800.124,A -85,B 0,C 180,E1 -23096.282,E2 -23096.282} C_VEL
LIN {X 0,Y 178.481,Z 810.126,A -85,B 0,C 180,E1 -23098.554,E2 -23098.554} C_VEL
LIN {X 0,Y 174.969,Z 819.148,A -85,B 0,C 180,E1 -23101.186,E2 -23101.186} C_VEL
LIN {X 0,Y 171.469,Z 827.679,A -85,B 0,C 180,E1 -23104.384,E2 -23104.384} C_VEL
LIN {X 0,Y 168.795,Z 833.898,A -85,B 0,C 180,E1 -23107.35,E2 -23107.35} C_VEL
LIN {X 0,Y 166.612,Z 838.841,A -85,B 0,C 180,E1 -23110.281,E2 -23110.281} C_VEL
LIN {X 0,Y 164.461,Z 843.625,A -85,B 0,C 180,E1 -23113.875,E2 -23113.875} C_VEL
LIN {X 0,Y 163.108,Z 847.289,A -85,B 0,C 180,E1 -23117.561,E2 -23117.561} C_VEL
LIN {X 0,Y 162.447,Z 849.177,A -85,B 0,C 180,E1 -23120.037,E2 -23120.037} C_VEL
LIN {X 0,Y 162.038,Z 850.6,A -85,B 0,C 180,E1 -23122.526,E2 -23122.526} C_VEL
LIN {X 0,Y 161.873,Z 852.116,A -85,B 0,C 180,E1 -23126.954,E2 -23126.954} C_VEL
LIN {X 0,Y 161.998,Z 852.444,A -85,B 0,C 180,E1 -23130.002,E2 -23130.002} C_VEL
LIN {X 0,Y 161.893,Z 852.076,A -85,B 0,C 180,E1 -23133.177,E2 -23133.177} C_VEL
LIN {X 0,Y 162.041,Z 850.564,A -85,B 0,C 180,E1 -23137.478,E2 -23137.478} C_VEL
LIN {X 0,Y 162.45,Z 849.121,A -85,B 0,C 180,E1 -23139.967,E2 -23139.967} C_VEL
LIN {X 0,Y 163.472,Z 846.134,A -85,B 0,C 180,E1 -23143.679,E2 -23143.679} C_VEL
LIN {X 0,Y 165.054,Z 842.086,A -85,B 0,C 180,E1 -23147.343,E2 -23147.343} C_VEL
LIN {X 0,Y 167.816,Z 835.854,A -85,B 0,C 180,E1 -23151.498,E2 -23151.498} C_VEL
LIN {X 0,Y 170.969,Z 828.807,A -85,B 0,C 180,E1 -23155.057,E2 -23155.057} C_VEL
LIN {X 0,Y 174.256,Z 820.562,A -85,B 0,C 180,E1 -23158.289,E2 -23158.289} C_VEL
LIN {X 0,Y 177.711,Z 811.824,A -85,B 0,C 180,E1 -23160.94,E2 -23160.94} C_VEL
LIN {X 0,Y 181.541,Z 801.062,A -85,B 0,C 180,E1 -23163.483,E2 -23163.483} C_VEL
LIN {X 0,Y 184.88,Z 790.184,A -85,B 0,C 180,E1 -23165.432,E2 -23165.432} C_VEL
LIN {X 0,Y 187.937,Z 778.022,A -85,B 0,C 180,E1 -23167.087,E2 -23167.087} C_VEL
LIN {X 0,Y 190.27,Z 766.528,A -85,B 0,C 180,E1 -23168.222,E2 -23168.222} C_VEL
LIN {X 0,Y 192.241,Z 753.447,A -85,B 0,C 180,E1 -23169.076,E2 -23169.076} C_VEL
LIN {X 0,Y 193.414,Z 737.849,A -85,B 0,C 180,E1 -23169.705,E2 -23169.705} C_VEL
LIN {X 0,Y 195.772,Z 694.159,A -85,B 0,C 180,E1 -23171.182,E2 -23171.182} C_VEL
LIN {X 0,Y 194.366,Z 670.116,A -85,B 0,C 180,E1 -23172.713,E2 -23172.713} C_VEL
LIN {X 0,Y 192.241,Z 646.814,A -85,B 0,C 180,E1 -23174.477,E2 -23174.477} C_VEL
LIN {X 0,Y 191.194,Z 638.072,A -85,B 0,C 180,E1 -23175.238,E2 -23175.238} C_VEL
LIN {X 0,Y 189.151,Z 632.305,A -85,B 0,C 180,E1 -23176.262,E2 -23176.262} C_VEL
LIN {X 0,Y 187.07,Z 620.424,A -85,B 0,C 180,E1 -23179.603,E2 -23179.603} C_VEL
LIN {X 0,Y 184.762,Z 615.21,A -85,B 0,C 180,E1 -23181.738,E2 -23181.738} C_VEL
LIN {X 0,Y 180.583,Z 607.284,A -85,B 0,C 180,E1 -23185.645,E2 -23185.645} C_VEL
LIN {X 0,Y 178.45,Z 603.294,A -85,B 0,C 180,E1 -23187.851,E2 -23187.851} C_VEL
LIN {X 0,Y 177.26,Z 601.799,A -85,B 0,C 180,E1 -23188.974,E2 -23188.974} C_VEL
LIN {X 0,Y 175.51,Z 598.26,A -85,B 0,C 180,E1 -23191.281,E2 -23191.281} C_VEL
LIN {X 0,Y 173.836,Z 595.068,A -85,B 0,C 180,E1 -23193.595,E2 -23193.595} C_VEL
LIN {X 0,Y 172.044,Z 592.946,A -85,B 0,C 180,E1 -23195.889,E2 -23195.889} C_VEL
LIN {X 0,Y 170.815,Z 590.239,A -85,B 0,C 180,E1 -23198.266,E2 -23198.266} C_VEL
LIN {X 0,Y 167.734,Z 585.068,A -85,B 0,C 180,E1 -23205.44,E2 -23205.44} C_VEL
LIN {X 0,Y 165.703,Z 582.572,A -85,B 0,C 180,E1 -23212.69,E2 -23212.69} C_VEL
LIN {X 0,Y 165.482,Z 581.585,A -85,B 0,C 180,E1 -23217.566,E2 -23217.566} C_VEL
LIN {X 0,Y 165.72,Z 581.566,A -85,B 0,C 180,E1 -23220,E2 -23220} C_VEL
LIN {X 0,Y 167.295,Z 584.482,A -85,B 0,C 180,E1 -23229.674,E2 -23229.674} C_VEL
LIN {X 0,Y 167.937,Z 585.883,A -85,B 0,C 180,E1 -23232.078,E2 -23232.078} C_VEL
LIN {X 0,Y 169.744,Z 589.272,A -85,B 0,C 180,E1 -23236.848,E2 -23236.848} C_VEL
LIN {X 0,Y 171.944,Z 593.779,A -85,B 0,C 180,E1 -23241.584,E2 -23241.584} C_VEL
LIN {X 0,Y 174.492,Z 599.301,A -85,B 0,C 180,E1 -23246.299,E2 -23246.299} C_VEL
LIN {X 0,Y 176.642,Z 604.121,A -85,B 0,C 180,E1 -23249.824,E2 -23249.824} C_VEL
LIN {X 0,Y 179.754,Z 612.378,A -85,B 0,C 180,E1 -23254.808,E2 -23254.808} C_VEL
LIN {X 0,Y 182.302,Z 619.957,A -85,B 0,C 180,E1 -23258.717,E2 -23258.717} C_VEL
LIN {X 0,Y 184.705,Z 628.252,A -85,B 0,C 180,E1 -23262.331,E2 -23262.331} C_VEL
LIN {X 0,Y 189.675,Z 637.821,A -85,B 0,C 180,E1 -23264.47,E2 -23264.47} C_VEL
LIN {X 0,Y 194.334,Z 648.251,A -85,B 0,C 180,E1 -23266.383,E2 -23266.383} C_VEL
LIN {X 0,Y 195.185,Z 650.503,A -85,B 0,C 180,E1 -23266.733,E2 -23266.733} C_VEL
LIN {X 0,Y 197.479,Z 672.219,A -85,B 0,C 180,E1 -23268.406,E2 -23268.406} C_VEL
LIN {X 0,Y 193.482,Z 740.237,A -85,B 0,C 180,E1 -23270.697,E2 -23270.697} C_VEL
LIN {X 0,Y 192.034,Z 753.034,A -85,B 0,C 180,E1 -23271.441,E2 -23271.441} C_VEL
LIN {X 0,Y 189.937,Z 765.31,A -85,B 0,C 180,E1 -23272.538,E2 -23272.538} C_VEL
LIN {X 0,Y 187.139,Z 777.677,A -85,B 0,C 180,E1 -23274.068,E2 -23274.068} C_VEL
LIN {X 0,Y 184.217,Z 788.039,A -85,B 0,C 180,E1 -23275.754,E2 -23275.754} C_VEL
LIN {X 0,Y 180.761,Z 798.653,A -85,B 0,C 180,E1 -23278.01,E2 -23278.01} C_VEL
LIN {X 0,Y 177.606,Z 807.319,A -85,B 0,C 180,E1 -23280.354,E2 -23280.354} C_VEL
LIN {X 0,Y 173.868,Z 816.716,A -85,B 0,C 180,E1 -23283.598,E2 -23283.598} C_VEL
LIN {X 0,Y 170.532,Z 824.185,A -85,B 0,C 180,E1 -23286.949,E2 -23286.949} C_VEL
LIN {X 0,Y 167.678,Z 830.181,A -85,B 0,C 180,E1 -23290.407,E2 -23290.407} C_VEL
LIN {X 0,Y 165.489,Z 834.913,A -85,B 0,C 180,E1 -23293.974,E2 -23293.974} C_VEL
LIN {X 0,Y 163.872,Z 838.527,A -85,B 0,C 180,E1 -23297.616,E2 -23297.616} C_VEL
LIN {X 0,Y 163.084,Z 840.387,A -85,B 0,C 180,E1 -23300.072,E2 -23300.072} C_VEL
LIN {X 0,Y 162.548,Z 841.801,A -85,B 0,C 180,E1 -23302.545,E2 -23302.545} C_VEL
LIN {X 0,Y 161.955,Z 843.405,A -85,B 0,C 180,E1 -23307.511,E2 -23307.511} C_VEL
LIN {X 0,Y 161.942,Z 843.633,A -85,B 0,C 180,E1 -23309.998,E2 -23309.998} C_VEL
LIN {X 0,Y 162.001,Z 843.19,A -85,B 0,C 180,E1 -23313.799,E2 -23313.799} C_VEL
LIN {X 0,Y 162.546,Z 841.876,A -85,B 0,C 180,E1 -23317.451,E2 -23317.451} C_VEL
LIN {X 0,Y 163.08,Z 840.504,A -85,B 0,C 180,E1 -23319.924,E2 -23319.924} C_VEL
LIN {X 0,Y 164.324,Z 837.619,A -85,B 0,C 180,E1 -23323.603,E2 -23323.603} C_VEL
LIN {X 0,Y 166.124,Z 833.693,A -85,B 0,C 180,E1 -23327.223,E2 -23327.223} C_VEL
LIN {X 0,Y 168.497,Z 828.607,A -85,B 0,C 180,E1 -23330.762,E2 -23330.762} C_VEL
LIN {X 0,Y 171.516,Z 822.19,A -85,B 0,C 180,E1 -23334.187,E2 -23334.187} C_VEL
LIN {X 0,Y 174.902,Z 814.408,A -85,B 0,C 180,E1 -23337.429,E2 -23337.429} C_VEL
LIN {X 0,Y 178.477,Z 805.209,A -85,B 0,C 180,E1 -23340.428,E2 -23340.428} C_VEL
LIN {X 0,Y 182.18,Z 794.811,A -85,B 0,C 180,E1 -23343.015,E2 -23343.015} C_VEL
LIN {X 0,Y 185.408,Z 784.619,A -85,B 0,C 180,E1 -23344.979,E2 -23344.979} C_VEL
LIN {X 0,Y 188.313,Z 773.407,A -85,B 0,C 180,E1 -23346.662,E2 -23346.662} C_VEL
LIN {X 0,Y 190.896,Z 760.665,A -85,B 0,C 180,E1 -23348.07,E2 -23348.07} C_VEL
LIN {X 0,Y 192.905,Z 747.637,A -85,B 0,C 180,E1 -23349.052,E2 -23349.052} C_VEL
LIN {X 0,Y 194.057,Z 734.839,A -85,B 0,C 180,E1 -23349.65,E2 -23349.65} C_VEL
LIN {X 0,Y 195.717,Z 704.018,A -85,B 0,C 180,E1 -23350.701,E2 -23350.701} C_VEL
LIN {X 0,Y 191.944,Z 706.535,A -85,B 0,C 180,E1 -23351.555,E2 -23351.555} C_VEL
LIN {X 0,Y 189.196,Z 707.536,A -85,B 0,C 180,E1 -23352.248,E2 -23352.248} C_VEL
LIN {X 0,Y 185.321,Z 712.003,A -85,B 0,C 180,E1 -23353.114,E2 -23353.114} C_VEL
LIN {X 0,Y 182.151,Z 714.182,A -85,B 0,C 180,E1 -23353.94,E2 -23353.94} C_VEL
LIN {X 0,Y 180.026,Z 714.756,A -85,B 0,C 180,E1 -23354.564,E2 -23354.564} C_VEL
LIN {X 0,Y 177.673,Z 715.158,A -85,B 0,C 180,E1 -23355.296,E2 -23355.296} C_VEL
LIN {X 0,Y 174.513,Z 718.676,A -85,B 0,C 180,E1 -23356.15,E2 -23356.15} C_VEL
LIN {X 0,Y 172.197,Z 720.149,A -85,B 0,C 180,E1 -23356.872,E2 -23356.872} C_VEL
LIN {X 0,Y 170.698,Z 720.22,A -85,B 0,C 180,E1 -23357.408,E2 -23357.408} C_VEL
LIN {X 0,Y 169.605,Z 719.234,A -85,B 0,C 180,E1 -23357.873,E2 -23357.873} C_VEL
LIN {X 0,Y 169.213,Z 717.172,A -85,B 0,C 180,E1 -23358.154,E2 -23358.154} C_VEL
LIN {X 0,Y 167.751,Z 727.968,A -85,B 0,C 180,E1 -23361.065,E2 -23361.065} C_VEL
LIN {X 0,Y 166.327,Z 738.106,A -85,B 0,C 180,E1 -23364.479,E2 -23364.479} C_VEL
LIN {X 0,Y 165.379,Z 746.979,A -85,B 0,C 180,E1 -23368.198,E2 -23368.198} C_VEL
LIN {X 0,Y 164.761,Z 754.264,A -85,B 0,C 180,E1 -23372.016,E2 -23372.016} C_VEL
LIN {X 0,Y 164.677,Z 760.463,A -85,B 0,C 180,E1 -23376.081,E2 -23376.081} C_VEL
LIN {X 0,Y 165.203,Z 765.253,A -85,B 0,C 180,E1 -23380.103,E2 -23380.103} C_VEL
LIN {X 0,Y 165.941,Z 767.738,A -85,B 0,C 180,E1 -23382.754,E2 -23382.754} C_VEL
LIN {X 0,Y 167.008,Z 769.725,A -85,B 0,C 180,E1 -23385.427,E2 -23385.427} C_VEL
LIN {X 0,Y 168.303,Z 771.187,A -85,B 0,C 180,E1 -23387.948,E2 -23387.948} C_VEL
LIN {X 0,Y 170.555,Z 772.456,A -85,B 0,C 180,E1 -23391.459,E2 -23391.459} C_VEL
LIN {X 0,Y 173.862,Z 772.812,A -85,B 0,C 180,E1 -23395.363,E2 -23395.363} C_VEL
LIN {X 0,Y 176.26,Z 772.422,A -85,B 0,C 180,E1 -23397.715,E2 -23397.715} C_VEL
LIN {X 0,Y 178.909,Z 771.606,A -85,B 0,C 180,E1 -23400,E2 -23400} C_VEL
LIN {X 0,Y 182.979,Z 769.706,A -85,B 0,C 180,E1 -23403.053,E2 -23403.053} C_VEL
LIN {X 0,Y 188.281,Z 766.33,A -85,B 0,C 180,E1 -23406.429,E2 -23406.429} C_VEL
LIN {X 0,Y 193.754,Z 762.013,A -85,B 0,C 180,E1 -23409.394,E2 -23409.394} C_VEL
LIN {X 0,Y 199.694,Z 756.335,A -85,B 0,C 180,E1 -23412.19,E2 -23412.19} C_VEL
LIN {X 0,Y 205.847,Z 749.287,A -85,B 0,C 180,E1 -23414.837,E2 -23414.837} C_VEL
LIN {X 0,Y 211.335,Z 742.064,A -85,B 0,C 180,E1 -23416.917,E2 -23416.917} C_VEL
LIN {X 0,Y 217,Z 733.321,A -85,B 0,C 180,E1 -23418.897,E2 -23418.897} C_VEL
LIN {X 0,Y 223.374,Z 721.457,A -85,B 0,C 180,E1 -23420.971,E2 -23420.971} C_VEL
LIN {X 0,Y 228.067,Z 710.737,A -85,B 0,C 180,E1 -23422.418,E2 -23422.418} C_VEL
LIN {X 0,Y 232.324,Z 698.345,A -85,B 0,C 180,E1 -23423.716,E2 -23423.716} C_VEL
LIN {X 0,Y 235.597,Z 685.521,A -85,B 0,C 180,E1 -23424.774,E2 -23424.774} C_VEL
LIN {X 0,Y 238.252,Z 670.672,A -85,B 0,C 180,E1 -23425.658,E2 -23425.658} C_VEL
LIN {X 0,Y 239.117,Z 665.16,A -85,B 0,C 180,E1 -23425.989,E2 -23425.989} C_VEL
LIN {X 0,Y 238.039,Z 664.136,A -85,B 0,C 180,E1 -23427.662,E2 -23427.662} C_VEL
LIN {X 0,Y 236.557,Z 664.345,A -85,B 0,C 180,E1 -23431.684,E2 -23431.684} C_VEL
LIN {X 0,Y 236.205,Z 666.545,A -85,B 0,C 180,E1 -23434.194,E2 -23434.194} C_VEL
LIN {X 0,Y 236.417,Z 671.982,A -85,B 0,C 180,E1 -23437.442,E2 -23437.442} C_VEL
LIN {X 0,Y 236.326,Z 674.153,A -85,B 0,C 180,E1 -23437.983,E2 -23437.983} C_VEL
LIN {X 0,Y 235.842,Z 677.707,A -85,B 0,C 180,E1 -23438.341,E2 -23438.341} C_VEL
LIN {X 0,Y 235.264,Z 680.931,A -85,B 0,C 180,E1 -23438.469,E2 -23438.469} C_VEL
LIN {X 0,Y 233.455,Z 690.187,A -85,B 0,C 180,E1 -23438.683,E2 -23438.683} C_VEL
LIN {X 0,Y 233.098,Z 692.234,A -85,B 0,C 180,E1 -23438.834,E2 -23438.834} C_VEL
LIN {X 0,Y 231.169,Z 701.426,A -85,B 0,C 180,E1 -23439.496,E2 -23439.496} C_VEL
LIN {X 0,Y 226.735,Z 715.963,A -85,B 0,C 180,E1 -23440.248,E2 -23440.248} C_VEL
LIN {X 0,Y 220.858,Z 730.413,A -85,B 0,C 180,E1 -23441.259,E2 -23441.259} C_VEL
LIN {X 0,Y 214.414,Z 743.179,A -85,B 0,C 180,E1 -23442.485,E2 -23442.485} C_VEL
LIN {X 0,Y 206.842,Z 755.786,A -85,B 0,C 180,E1 -23444.132,E2 -23444.132} C_VEL
LIN {X 0,Y 199.659,Z 766.108,A -85,B 0,C 180,E1 -23445.96,E2 -23445.96} C_VEL
LIN {X 0,Y 192.218,Z 775.434,A -85,B 0,C 180,E1 -23448.147,E2 -23448.147} C_VEL
LIN {X 0,Y 185.328,Z 783.239,A -85,B 0,C 180,E1 -23450.569,E2 -23450.569} C_VEL
LIN {X 0,Y 180.125,Z 788.749,A -85,B 0,C 180,E1 -23452.791,E2 -23452.791} C_VEL
LIN {X 0,Y 179.387,Z 789.629,A -85,B 0,C 180,E1 -23453.139,E2 -23453.139} C_VEL
LIN {X 0,Y 176.114,Z 799.946,A -85,B 0,C 180,E1 -23454.998,E2 -23454.998} C_VEL
LIN {X 0,Y 172.435,Z 809.943,A -85,B 0,C 180,E1 -23457.317,E2 -23457.317} C_VEL
LIN {X 0,Y 168.757,Z 818.962,A -85,B 0,C 180,E1 -23460.02,E2 -23460.02} C_VEL
LIN {X 0,Y 164.787,Z 828.129,A -85,B 0,C 180,E1 -23463.589,E2 -23463.589} C_VEL
LIN {X 0,Y 161.719,Z 834.789,A -85,B 0,C 180,E1 -23466.978,E2 -23466.978} C_VEL
LIN {X 0,Y 159.069,Z 840.385,A -85,B 0,C 180,E1 -23470.651,E2 -23470.651} C_VEL
LIN {X 0,Y 157.03,Z 844.777,A -85,B 0,C 180,E1 -23474.425,E2 -23474.425} C_VEL
LIN {X 0,Y 156.132,Z 847.096,A -85,B 0,C 180,E1 -23476.996,E2 -23476.996} C_VEL
LIN {X 0,Y 155.443,Z 848.984,A -85,B 0,C 180,E1 -23479.583,E2 -23479.583} C_VEL
LIN {X 0,Y 154.981,Z 850.407,A -85,B 0,C 180,E1 -23482.183,E2 -23482.183} C_VEL
LIN {X 0,Y 154.792,Z 852.008,A -85,B 0,C 180,E1 -23487.268,E2 -23487.268} C_VEL
LIN {X 0,Y 154.908,Z 852.251,A -85,B 0,C 180,E1 -23490.002,E2 -23490.002} C_VEL
LIN {X 0,Y 154.81,Z 851.969,A -85,B 0,C 180,E1 -23492.868,E2 -23492.868} C_VEL
LIN {X 0,Y 154.984,Z 850.371,A -85,B 0,C 180,E1 -23497.821,E2 -23497.821} C_VEL
LIN {X 0,Y 155.445,Z 848.928,A -85,B 0,C 180,E1 -23500.421,E2 -23500.421} C_VEL
LIN {X 0,Y 156.54,Z 845.939,A -85,B 0,C 180,E1 -23504.298,E2 -23504.298} C_VEL
LIN {X 0,Y 158.279,Z 841.893,A -85,B 0,C 180,E1 -23508.11,E2 -23508.11} C_VEL
LIN {X 0,Y 161.192,Z 835.66,A -85,B 0,C 180,E1 -23512.429,E2 -23512.429} C_VEL
LIN {X 0,Y 164.276,Z 829.177,A -85,B 0,C 180,E1 -23515.84,E2 -23515.84} C_VEL
LIN {X 0,Y 167.344,Z 821.93,A -85,B 0,C 180,E1 -23518.881,E2 -23518.881} C_VEL
LIN {X 0,Y 170.878,Z 813.56,A -85,B 0,C 180,E1 -23521.629,E2 -23521.629} C_VEL
LIN {X 0,Y 174.822,Z 803.199,A -85,B 0,C 180,E1 -23524.252,E2 -23524.252} C_VEL
LIN {X 0,Y 178.688,Z 791.539,A -85,B 0,C 180,E1 -23526.506,E2 -23526.506} C_VEL
LIN {X 0,Y 181.835,Z 779.79,A -85,B 0,C 180,E1 -23528.202,E2 -23528.202} C_VEL
LIN {X 0,Y 184.503,Z 767.627,A -85,B 0,C 180,E1 -23529.47,E2 -23529.47} C_VEL
LIN {X 0,Y 186.594,Z 755.123,A -85,B 0,C 180,E1 -23530.349,E2 -23530.349} C_VEL
LIN {X 0,Y 187.794,Z 741.237,A -85,B 0,C 180,E1 -23530.971,E2 -23530.971} C_VEL
LIN {X 0,Y 190.441,Z 694.808,A -85,B 0,C 180,E1 -23532.563,E2 -23532.563} C_VEL
LIN {X 0,Y 189.159,Z 671.237,A -85,B 0,C 180,E1 -23534.124,E2 -23534.124} C_VEL
LIN {X 0,Y 187.39,Z 650.196,A -85,B 0,C 180,E1 -23535.766,E2 -23535.766} C_VEL
LIN {X 0,Y 186.351,Z 640.933,A -85,B 0,C 180,E1 -23536.598,E2 -23536.598} C_VEL
LIN {X 0,Y 183.231,Z 632.117,A -85,B 0,C 180,E1 -23538.233,E2 -23538.233} C_VEL
LIN {X 0,Y 181.967,Z 624.382,A -85,B 0,C 180,E1 -23540.576,E2 -23540.576} C_VEL
LIN {X 0,Y 179.043,Z 617.961,A -85,B 0,C 180,E1 -23543.41,E2 -23543.41} C_VEL
LIN {X 0,Y 174.288,Z 608.82,A -85,B 0,C 180,E1 -23548.385,E2 -23548.385} C_VEL
LIN {X 0,Y 173.125,Z 607.326,A -85,B 0,C 180,E1 -23549.507,E2 -23549.507} C_VEL
LIN {X 0,Y 171.553,Z 603.999,A -85,B 0,C 180,E1 -23551.699,E2 -23551.699} C_VEL
LIN {X 0,Y 169.722,Z 600.674,A -85,B 0,C 180,E1 -23554.228,E2 -23554.228} C_VEL
LIN {X 0,Y 166.789,Z 595.893,A -85,B 0,C 180,E1 -23559.012,E2 -23559.012} C_VEL
LIN {X 0,Y 164.167,Z 591.442,A -85,B 0,C 180,E1 -23565.116,E2 -23565.116} C_VEL
LIN {X 0,Y 162.146,Z 588.769,A -85,B 0,C 180,E1 -23572.529,E2 -23572.529} C_VEL
LIN {X 0,Y 161.891,Z 587.743,A -85,B 0,C 180,E1 -23577.512,E2 -23577.512} C_VEL
LIN {X 0,Y 162.062,Z 587.66,A -85,B 0,C 180,E1 -23580,E2 -23580} C_VEL
LIN {X 0,Y 163.494,Z 590.637,A -85,B 0,C 180,E1 -23589.901,E2 -23589.901} C_VEL
LIN {X 0,Y 165.817,Z 595.642,A -85,B 0,C 180,E1 -23597.259,E2 -23597.259} C_VEL
LIN {X 0,Y 167.898,Z 600.202,A -85,B 0,C 180,E1 -23602.131,E2 -23602.131} C_VEL
LIN {X 0,Y 170.49,Z 605.804,A -85,B 0,C 180,E1 -23606.965,E2 -23606.965} C_VEL
LIN {X 0,Y 172.941,Z 612.317,A -85,B 0,C 180,E1 -23611.414,E2 -23611.414} C_VEL
LIN {X 0,Y 175.55,Z 619.715,A -85,B 0,C 180,E1 -23615.767,E2 -23615.767} C_VEL
LIN {X 0,Y 177.915,Z 627.574,A -85,B 0,C 180,E1 -23619.678,E2 -23619.678} C_VEL
LIN {X 0,Y 178.816,Z 629.545,A -85,B 0,C 180,E1 -23620.288,E2 -23620.288} C_VEL
LIN {X 0,Y 184.065,Z 639.415,A -85,B 0,C 180,E1 -23622.746,E2 -23622.746} C_VEL
LIN {X 0,Y 189.046,Z 650.294,A -85,B 0,C 180,E1 -23624.939,E2 -23624.939} C_VEL
LIN {X 0,Y 190.25,Z 653.807,A -85,B 0,C 180,E1 -23625.485,E2 -23625.485} C_VEL
LIN {X 0,Y 192.163,Z 672.847,A -85,B 0,C 180,E1 -23627.009,E2 -23627.009} C_VEL
LIN {X 0,Y 188.178,Z 739.028,A -85,B 0,C 180,E1 -23629.274,E2 -23629.274} C_VEL
LIN {X 0,Y 186.67,Z 752.36,A -85,B 0,C 180,E1 -23630.028,E2 -23630.028} C_VEL
LIN {X 0,Y 184.577,Z 764.404,A -85,B 0,C 180,E1 -23631.077,E2 -23631.077} C_VEL
LIN {X 0,Y 181.881,Z 776.152,A -85,B 0,C 180,E1 -23632.511,E2 -23632.511} C_VEL
LIN {X 0,Y 178.406,Z 788.224,A -85,B 0,C 180,E1 -23634.474,E2 -23634.474} C_VEL
LIN {X 0,Y 174.79,Z 798.841,A -85,B 0,C 180,E1 -23636.779,E2 -23636.779} C_VEL
LIN {X 0,Y 170.964,Z 808.768,A -85,B 0,C 180,E1 -23639.574,E2 -23639.574} C_VEL
LIN {X 0,Y 167.536,Z 816.907,A -85,B 0,C 180,E1 -23642.518,E2 -23642.518} C_VEL
LIN {X 0,Y 164.034,Z 824.376,A -85,B 0,C 180,E1 -23645.98,E2 -23645.98} C_VEL
LIN {X 0,Y 160.991,Z 830.374,A -85,B 0,C 180,E1 -23649.557,E2 -23649.557} C_VEL
LIN {X 0,Y 158.682,Z 835.106,A -85,B 0,C 180,E1 -23653.267,E2 -23653.267} C_VEL
LIN {X 0,Y 156.927,Z 838.721,A -85,B 0,C 180,E1 -23657.058,E2 -23657.058} C_VEL
LIN {X 0,Y 156.085,Z 840.58,A -85,B 0,C 180,E1 -23659.622,E2 -23659.622} C_VEL
LIN {X 0,Y 155.506,Z 841.995,A -85,B 0,C 180,E1 -23662.206,E2 -23662.206} C_VEL
LIN {X 0,Y 154.865,Z 843.598,A -85,B 0,C 180,E1 -23667.397,E2 -23667.397} C_VEL
LIN {X 0,Y 154.854,Z 843.826,A -85,B 0,C 180,E1 -23669.998,E2 -23669.998} C_VEL
LIN {X 0,Y 154.859,Z 843.521,A -85,B 0,C 180,E1 -23673.207,E2 -23673.207} C_VEL
LIN {X 0,Y 155.504,Z 842.069,A -85,B 0,C 180,E1 -23677.79,E2 -23677.79} C_VEL
LIN {X 0,Y 156.081,Z 840.696,A -85,B 0,C 180,E1 -23680.374,E2 -23680.374} C_VEL
LIN {X 0,Y 157.422,Z 837.811,A -85,B 0,C 180,E1 -23684.212,E2 -23684.212} C_VEL
LIN {X 0,Y 159.363,Z 833.884,A -85,B 0,C 180,E1 -23687.979,E2 -23687.979} C_VEL
LIN {X 0,Y 161.885,Z 828.796,A -85,B 0,C 180,E1 -23691.652,E2 -23691.652} C_VEL
LIN {X 0,Y 165.075,Z 822.378,A -85,B 0,C 180,E1 -23695.195,E2 -23695.195} C_VEL
LIN {X 0,Y 168.496,Z 814.875,A -85,B 0,C 180,E1 -23698.434,E2 -23698.434} C_VEL
LIN {X 0,Y 172.082,Z 806.214,A -85,B 0,C 180,E1 -23701.377,E2 -23701.377} C_VEL
LIN {X 0,Y 175.898,Z 796.132,A -85,B 0,C 180,E1 -23704.009,E2 -23704.009} C_VEL
LIN {X 0,Y 179.642,Z 784.793,A -85,B 0,C 180,E1 -23706.276,E2 -23706.276} C_VEL
LIN {X 0,Y 182.676,Z 773.573,A -85,B 0,C 180,E1 -23707.99,E2 -23707.99} C_VEL
LIN {X 0,Y 185.367,Z 760.819,A -85,B 0,C 180,E1 -23709.421,E2 -23709.421} C_VEL
LIN {X 0,Y 187.438,Z 747.814,A -85,B 0,C 180,E1 -23710.417,E2 -23710.417} C_VEL
LIN {X 0,Y 188.648,Z 735.031,A -85,B 0,C 180,E1 -23711.019,E2 -23711.019} C_VEL
LIN {X 0,Y 189.695,Z 715.961,A -85,B 0,C 180,E1 -23711.69,E2 -23711.69} C_VEL
LIN {X 0,Y 185.578,Z 719.538,A -85,B 0,C 180,E1 -23712.649,E2 -23712.649} C_VEL
LIN {X 0,Y 181.983,Z 721.35,A -85,B 0,C 180,E1 -23713.605,E2 -23713.605} C_VEL
LIN {X 0,Y 179.24,Z 722.052,A -85,B 0,C 180,E1 -23714.409,E2 -23714.409} C_VEL
LIN {X 0,Y 175.69,Z 725.339,A -85,B 0,C 180,E1 -23715.369,E2 -23715.369} C_VEL
LIN {X 0,Y 172.793,Z 726.975,A -85,B 0,C 180,E1 -23716.256,E2 -23716.256} C_VEL
LIN {X 0,Y 169.757,Z 727.331,A -85,B 0,C 180,E1 -23717.317,E2 -23717.317} C_VEL
LIN {X 0,Y 168.732,Z 727.196,A -85,B 0,C 180,E1 -23717.705,E2 -23717.705} C_VEL
LIN {X 0,Y 165.502,Z 730.301,A -85,B 0,C 180,E1 -23718.751,E2 -23718.751} C_VEL
LIN {X 0,Y 163.497,Z 731.367,A -85,B 0,C 180,E1 -23719.489,E2 -23719.489} C_VEL
LIN {X 0,Y 161.599,Z 731.146,A -85,B 0,C 180,E1 -23720.3,E2 -23720.3} C_VEL
LIN {X 0,Y 160.772,Z 729.583,A -85,B 0,C 180,E1 -23720.766,E2 -23720.766} C_VEL
LIN {X 0,Y 160.644,Z 728.525,A -85,B 0,C 180,E1 -23720.93,E2 -23720.93} C_VEL
LIN {X 0,Y 159.288,Z 738.031,A -85,B 0,C 180,E1 -23724.224,E2 -23724.224} C_VEL
LIN {X 0,Y 158.353,Z 746.488,A -85,B 0,C 180,E1 -23727.82,E2 -23727.82} C_VEL
LIN {X 0,Y 157.656,Z 754.479,A -85,B 0,C 180,E1 -23732.008,E2 -23732.008} C_VEL
LIN {X 0,Y 157.621,Z 760.987,A -85,B 0,C 180,E1 -23736.341,E2 -23736.341} C_VEL
LIN {X 0,Y 158.205,Z 765.893,A -85,B 0,C 180,E1 -23740.538,E2 -23740.538} C_VEL
LIN {X 0,Y 159.833,Z 770.068,A -85,B 0,C 180,E1 -23745.309,E2 -23745.309} C_VEL
LIN {X 0,Y 162.347,Z 772.738,A -85,B 0,C 180,E1 -23750.028,E2 -23750.028} C_VEL
LIN {X 0,Y 164.198,Z 773.618,A -85,B 0,C 180,E1 -23752.622,E2 -23752.622} C_VEL
LIN {X 0,Y 166.362,Z 774.047,A -85,B 0,C 180,E1 -23755.153,E2 -23755.153} C_VEL
LIN {X 0,Y 168.807,Z 773.983,A -85,B 0,C 180,E1 -23757.636,E2 -23757.636} C_VEL
LIN {X 0,Y 171.478,Z 773.505,A -85,B 0,C 180,E1 -23760,E2 -23760} C_VEL
LIN {X 0,Y 176.008,Z 771.917,A -85,B 0,C 180,E1 -23763.438,E2 -23763.438} C_VEL
LIN {X 0,Y 182.86,Z 768.192,A -85,B 0,C 180,E1 -23767.731,E2 -23767.731} C_VEL
LIN {X 0,Y 188.63,Z 764.03,A -85,B 0,C 180,E1 -23770.736,E2 -23770.736} C_VEL
LIN {X 0,Y 195.333,Z 758.219,A -85,B 0,C 180,E1 -23773.736,E2 -23773.736} C_VEL
LIN {X 0,Y 201.399,Z 751.858,A -85,B 0,C 180,E1 -23776.21,E2 -23776.21} C_VEL
LIN {X 0,Y 208.271,Z 743.323,A -85,B 0,C 180,E1 -23778.689,E2 -23778.689} C_VEL
LIN {X 0,Y 214.299,Z 734.618,A -85,B 0,C 180,E1 -23780.643,E2 -23780.643} C_VEL
LIN {X 0,Y 220.373,Z 723.939,A -85,B 0,C 180,E1 -23782.501,E2 -23782.501} C_VEL
LIN {X 0,Y 225.283,Z 713.496,A -85,B 0,C 180,E1 -23783.926,E2 -23783.926} C_VEL
LIN {X 0,Y 229.673,Z 701.995,A -85,B 0,C 180,E1 -23785.163,E2 -23785.163} C_VEL
LIN {X 0,Y 233.303,Z 689.393,A -85,B 0,C 180,E1 -23786.247,E2 -23786.247} C_VEL
LIN {X 0,Y 236.009,Z 675.854,A -85,B 0,C 180,E1 -23787.092,E2 -23787.092} C_VEL
LIN {X 0,Y 236.769,Z 671.213,A -85,B 0,C 180,E1 -23787.367,E2 -23787.367} C_VEL
LIN {X 0,Y 235.222,Z 671.139,A -85,B 0,C 180,E1 -23791.159,E2 -23791.159} C_VEL
LIN {X 0,Y 234.756,Z 672.802,A -85,B 0,C 180,E1 -23793.428,E2 -23793.428} C_VEL
LIN {X 0,Y 234.719,Z 678.641,A -85,B 0,C 180,E1 -23796.921,E2 -23796.921} C_VEL
LIN {X 0,Y 234.809,Z 680.871,A -85,B 0,C 180,E1 -23797.8,E2 -23797.8} C_VEL
LIN {X 0,Y 233.098,Z 692.234,A -85,B 0,C 180,E1 -23798.834,E2 -23798.834} C_VEL
LIN {X 0,Y 232.596,Z 694.735,A -85,B 0,C 180,E1 -23798.971,E2 -23798.971} C_VEL
LIN {X 0,Y 231.519,Z 698.548,A -85,B 0,C 180,E1 -23798.905,E2 -23798.905} C_VEL
LIN {X 0,Y 227.759,Z 708.523,A -85,B 0,C 180,E1 -23798.264,E2 -23798.264} C_VEL
LIN {X 0,Y 226.313,Z 712.304,A -85,B 0,C 180,E1 -23798.288,E2 -23798.288} C_VEL
LIN {X 0,Y 220.833,Z 725.892,A -85,B 0,C 180,E1 -23799.132,E2 -23799.132} C_VEL
LIN {X 0,Y 214.155,Z 739.236,A -85,B 0,C 180,E1 -23800.274,E2 -23800.274} C_VEL
LIN {X 0,Y 207.69,Z 750.149,A -85,B 0,C 180,E1 -23801.527,E2 -23801.527} C_VEL
LIN {X 0,Y 201.391,Z 759.306,A -85,B 0,C 180,E1 -23802.878,E2 -23802.878} C_VEL
LIN {X 0,Y 193.379,Z 769.492,A -85,B 0,C 180,E1 -23804.875,E2 -23804.875} C_VEL
LIN {X 0,Y 185.806,Z 778.042,A -85,B 0,C 180,E1 -23807.094,E2 -23807.094} C_VEL
LIN {X 0,Y 178.815,Z 785.134,A -85,B 0,C 180,E1 -23809.575,E2 -23809.575} C_VEL
LIN {X 0,Y 173.508,Z 790.232,A -85,B 0,C 180,E1 -23811.854,E2 -23811.854} C_VEL
LIN {X 0,Y 169.908,Z 800.999,A -85,B 0,C 180,E1 -23813.887,E2 -23813.887} C_VEL
LIN {X 0,Y 165.703,Z 811.692,A -85,B 0,C 180,E1 -23816.542,E2 -23816.542} C_VEL
LIN {X 0,Y 161.895,Z 820.391,A -85,B 0,C 180,E1 -23819.334,E2 -23819.334} C_VEL
LIN {X 0,Y 158.167,Z 828.5,A -85,B 0,C 180,E1 -23822.708,E2 -23822.708} C_VEL
LIN {X 0,Y 155.201,Z 834.6,A -85,B 0,C 180,E1 -23825.952,E2 -23825.952} C_VEL
LIN {X 0,Y 152.362,Z 840.194,A -85,B 0,C 180,E1 -23829.763,E2 -23829.763} C_VEL
LIN {X 0,Y 150.16,Z 844.584,A -85,B 0,C 180,E1 -23833.693,E2 -23833.693} C_VEL
LIN {X 0,Y 149.178,Z 846.903,A -85,B 0,C 180,E1 -23836.378,E2 -23836.378} C_VEL
LIN {X 0,Y 148.427,Z 848.791,A -85,B 0,C 180,E1 -23839.085,E2 -23839.085} C_VEL
LIN {X 0,Y 147.947,Z 850.214,A -85,B 0,C 180,E1 -23841.809,E2 -23841.809} C_VEL
LIN {X 0,Y 147.715,Z 851.84,A -85,B 0,C 180,E1 -23847.275,E2 -23847.275} C_VEL
LIN {X 0,Y 147.825,Z 852.058,A -85,B 0,C 180,E1 -23850.002,E2 -23850.002} C_VEL
LIN {X 0,Y 147.719,Z 851.825,A -85,B 0,C 180,E1 -23852.729,E2 -23852.729} C_VEL
LIN {X 0,Y 147.949,Z 850.177,A -85,B 0,C 180,E1 -23858.195,E2 -23858.195} C_VEL
LIN {X 0,Y 148.428,Z 848.733,A -85,B 0,C 180,E1 -23860.92,E2 -23860.92} C_VEL
LIN {X 0,Y 149.635,Z 845.745,A -85,B 0,C 180,E1 -23864.973,E2 -23864.973} C_VEL
LIN {X 0,Y 151.535,Z 841.7,A -85,B 0,C 180,E1 -23868.946,E2 -23868.946} C_VEL
LIN {X 0,Y 154.629,Z 835.467,A -85,B 0,C 180,E1 -23873.436,E2 -23873.436} C_VEL
LIN {X 0,Y 158.113,Z 828.422,A -85,B 0,C 180,E1 -23877.254,E2 -23877.254} C_VEL
LIN {X 0,Y 161.841,Z 820.179,A -85,B 0,C 180,E1 -23880.682,E2 -23880.682} C_VEL
LIN {X 0,Y 165.643,Z 811.444,A -85,B 0,C 180,E1 -23883.477,E2 -23883.477} C_VEL
LIN {X 0,Y 169.889,Z 800.69,A -85,B 0,C 180,E1 -23886.123,E2 -23886.123} C_VEL
LIN {X 0,Y 173.509,Z 789.819,A -85,B 0,C 180,E1 -23888.15,E2 -23888.15} C_VEL
LIN {X 0,Y 176.826,Z 777.669,A -85,B 0,C 180,E1 -23889.86,E2 -23889.86} C_VEL
LIN {X 0,Y 179.35,Z 766.192,A -85,B 0,C 180,E1 -23891.025,E2 -23891.025} C_VEL
LIN {X 0,Y 181.418,Z 753.571,A -85,B 0,C 180,E1 -23891.874,E2 -23891.874} C_VEL
LIN {X 0,Y 182.682,Z 737.972,A -85,B 0,C 180,E1 -23892.543,E2 -23892.543} C_VEL
LIN {X 0,Y 185.186,Z 695.147,A -85,B 0,C 180,E1 -23894.052,E2 -23894.052} C_VEL
LIN {X 0,Y 184.038,Z 671.44,A -85,B 0,C 180,E1 -23895.675,E2 -23895.675} C_VEL
LIN {X 0,Y 182.252,Z 649.109,A -85,B 0,C 180,E1 -23897.507,E2 -23897.507} C_VEL
LIN {X 0,Y 181.61,Z 643.766,A -85,B 0,C 180,E1 -23898.035,E2 -23898.035} C_VEL
LIN {X 0,Y 177.554,Z 632.349,A -85,B 0,C 180,E1 -23900.255,E2 -23900.255} C_VEL
LIN {X 0,Y 177.046,Z 629.069,A -85,B 0,C 180,E1 -23901.302,E2 -23901.302} C_VEL
LIN {X 0,Y 175.065,Z 624.323,A -85,B 0,C 180,E1 -23903.41,E2 -23903.41} C_VEL
LIN {X 0,Y 170.563,Z 615.348,A -85,B 0,C 180,E1 -23908.308,E2 -23908.308} C_VEL
LIN {X 0,Y 167.315,Z 609.275,A -85,B 0,C 180,E1 -23912.48,E2 -23912.48} C_VEL
LIN {X 0,Y 165.632,Z 606.276,A -85,B 0,C 180,E1 -23914.893,E2 -23914.893} C_VEL
LIN {X 0,Y 162.783,Z 601.52,A -85,B 0,C 180,E1 -23919.794,E2 -23919.794} C_VEL
LIN {X 0,Y 160.559,Z 597.835,A -85,B 0,C 180,E1 -23924.774,E2 -23924.774} C_VEL
LIN {X 0,Y 159.009,Z 595.7,A -85,B 0,C 180,E1 -23929.817,E2 -23929.817} C_VEL
LIN {X 0,Y 158.303,Z 593.889,A -85,B 0,C 180,E1 -23937.456,E2 -23937.456} C_VEL
LIN {X 0,Y 158.402,Z 593.771,A -85,B 0,C 180,E1 -23940,E2 -23940} C_VEL
LIN {X 0,Y 158.96,Z 595.773,A -85,B 0,C 180,E1 -23947.622,E2 -23947.622} C_VEL
LIN {X 0,Y 159.59,Z 596.742,A -85,B 0,C 180,E1 -23950.146,E2 -23950.146} C_VEL
LIN {X 0,Y 161.556,Z 601.215,A -85,B 0,C 180,E1 -23956.851,E2 -23956.851} C_VEL
LIN {X 0,Y 163.956,Z 606.673,A -85,B 0,C 180,E1 -23962.693,E2 -23962.693} C_VEL
LIN {X 0,Y 166.33,Z 612.295,A -85,B 0,C 180,E1 -23967.459,E2 -23967.459} C_VEL
LIN {X 0,Y 169.094,Z 620.062,A -85,B 0,C 180,E1 -23972.705,E2 -23972.705} C_VEL
LIN {X 0,Y 171.839,Z 628.58,A -85,B 0,C 180,E1 -23977.385,E2 -23977.385} C_VEL
LIN {X 0,Y 177.547,Z 639.007,A -85,B 0,C 180,E1 -23980.385,E2 -23980.385} C_VEL
LIN {X 0,Y 182.613,Z 649.51,A -85,B 0,C 180,E1 -23982.826,E2 -23982.826} C_VEL
LIN {X 0,Y 185.301,Z 656.164,A -85,B 0,C 180,E1 -23984.085,E2 -23984.085} C_VEL
LIN {X 0,Y 187.001,Z 673.902,A -85,B 0,C 180,E1 -23985.568,E2 -23985.568} C_VEL
LIN {X 0,Y 182.72,Z 740.747,A -85,B 0,C 180,E1 -23987.894,E2 -23987.894} C_VEL
LIN {X 0,Y 181.016,Z 754.108,A -85,B 0,C 180,E1 -23988.696,E2 -23988.696} C_VEL
LIN {X 0,Y 178.656,Z 766.741,A -85,B 0,C 180,E1 -23989.895,E2 -23989.895} C_VEL
LIN {X 0,Y 175.863,Z 778.039,A -85,B 0,C 180,E1 -23991.359,E2 -23991.359} C_VEL
LIN {X 0,Y 172.697,Z 788.408,A -85,B 0,C 180,E1 -23993.11,E2 -23993.11} C_VEL
LIN {X 0,Y 168.898,Z 799.029,A -85,B 0,C 180,E1 -23995.46,E2 -23995.46} C_VEL
LIN {X 0,Y 165.402,Z 807.699,A -85,B 0,C 180,E1 -23997.918,E2 -23997.918} C_VEL
LIN {X 0,Y 161.268,Z 817.099,A -85,B 0,C 180,E1 -24001.354,E2 -24001.354} C_VEL
LIN {X 0,Y 157.578,Z 824.568,A -85,B 0,C 180,E1 -24004.93,E2 -24004.93} C_VEL
LIN {X 0,Y 154.345,Z 830.567,A -85,B 0,C 180,E1 -24008.635,E2 -24008.635} C_VEL
LIN {X 0,Y 151.885,Z 835.3,A -85,B 0,C 180,E1 -24012.494,E2 -24012.494} C_VEL
LIN {X 0,Y 150.01,Z 838.914,A -85,B 0,C 180,E1 -24016.45,E2 -24016.45} C_VEL
LIN {X 0,Y 149.11,Z 840.774,A -85,B 0,C 180,E1 -24019.131,E2 -24019.131} C_VEL
LIN {X 0,Y 148.469,Z 842.188,A -85,B 0,C 180,E1 -24021.834,E2 -24021.834} C_VEL
LIN {X 0,Y 147.796,Z 843.79,A -85,B 0,C 180,E1 -24027.272,E2 -24027.272} C_VEL
LIN {X 0,Y 147.766,Z 844.019,A -85,B 0,C 180,E1 -24029.998,E2 -24029.998} C_VEL
LIN {X 0,Y 148.01,Z 843.233,A -85,B 0,C 180,E1 -24035.447,E2 -24035.447} C_VEL
LIN {X 0,Y 148.467,Z 842.261,A -85,B 0,C 180,E1 -24038.162,E2 -24038.162} C_VEL
LIN {X 0,Y 149.106,Z 840.888,A -85,B 0,C 180,E1 -24040.865,E2 -24040.865} C_VEL
LIN {X 0,Y 150.549,Z 838.002,A -85,B 0,C 180,E1 -24044.875,E2 -24044.875} C_VEL
LIN {X 0,Y 152.611,Z 834.075,A -85,B 0,C 180,E1 -24048.803,E2 -24048.803} C_VEL
LIN {X 0,Y 155.291,Z 828.986,A -85,B 0,C 180,E1 -24052.621,E2 -24052.621} C_VEL
LIN {X 0,Y 158.692,Z 822.566,A -85,B 0,C 180,E1 -24056.284,E2 -24056.284} C_VEL
LIN {X 0,Y 162.169,Z 815.301,A -85,B 0,C 180,E1 -24059.534,E2 -24059.534} C_VEL
LIN {X 0,Y 166.054,Z 806.396,A -85,B 0,C 180,E1 -24062.655,E2 -24062.655} C_VEL
LIN {X 0,Y 170.046,Z 796.312,A -85,B 0,C 180,E1 -24065.35,E2 -24065.35} C_VEL
LIN {X 0,Y 173.981,Z 784.968,A -85,B 0,C 180,E1 -24067.657,E2 -24067.657} C_VEL
LIN {X 0,Y 177.135,Z 773.74,A -85,B 0,C 180,E1 -24069.403,E2 -24069.403} C_VEL
LIN {X 0,Y 179.948,Z 760.972,A -85,B 0,C 180,E1 -24070.854,E2 -24070.854} C_VEL
LIN {X 0,Y 182.065,Z 748.212,A -85,B 0,C 180,E1 -24071.846,E2 -24071.846} C_VEL
LIN {X 0,Y 183.374,Z 734.763,A -85,B 0,C 180,E1 -24072.486,E2 -24072.486} C_VEL
LIN {X 0,Y 183.645,Z 727.804,A -85,B 0,C 180,E1 -24072.773,E2 -24072.773} C_VEL
LIN {X 0,Y 180.706,Z 728.906,A -85,B 0,C 180,E1 -24073.584,E2 -24073.584} C_VEL
LIN {X 0,Y 176.317,Z 732.368,A -85,B 0,C 180,E1 -24074.764,E2 -24074.764} C_VEL
LIN {X 0,Y 172.783,Z 733.959,A -85,B 0,C 180,E1 -24075.848,E2 -24075.848} C_VEL
LIN {X 0,Y 169.393,Z 734.668,A -85,B 0,C 180,E1 -24077.001,E2 -24077.001} C_VEL
LIN {X 0,Y 165.572,Z 737.479,A -85,B 0,C 180,E1 -24078.249,E2 -24078.249} C_VEL
LIN {X 0,Y 163.177,Z 738.381,A -85,B 0,C 180,E1 -24079.133,E2 -24079.133} C_VEL
LIN {X 0,Y 159.503,Z 738.269,A -85,B 0,C 180,E1 -24080.699,E2 -24080.699} C_VEL
LIN {X 0,Y 156.275,Z 740.717,A -85,B 0,C 180,E1 -24081.939,E2 -24081.939} C_VEL
LIN {X 0,Y 155.078,Z 741.2,A -85,B 0,C 180,E1 -24082.462,E2 -24082.462} C_VEL
LIN {X 0,Y 152.975,Z 740.929,A -85,B 0,C 180,E1 -24083.532,E2 -24083.532} C_VEL
LIN {X 0,Y 152.173,Z 739.159,A -85,B 0,C 180,E1 -24084.129,E2 -24084.129} C_VEL
LIN {X 0,Y 152.147,Z 738.608,A -85,B 0,C 180,E1 -24084.224,E2 -24084.224} C_VEL
LIN {X 0,Y 151.127,Z 748.113,A -85,B 0,C 180,E1 -24088.455,E2 -24088.455} C_VEL
LIN {X 0,Y 150.516,Z 755.441,A -85,B 0,C 180,E1 -24092.512,E2 -24092.512} C_VEL
LIN {X 0,Y 150.539,Z 761.425,A -85,B 0,C 180,E1 -24096.62,E2 -24096.62} C_VEL
LIN {X 0,Y 151.212,Z 766.506,A -85,B 0,C 180,E1 -24101.013,E2 -24101.013} C_VEL
LIN {X 0,Y 152.627,Z 770.273,A -85,B 0,C 180,E1 -24105.225,E2 -24105.225} C_VEL
LIN {X 0,Y 154.81,Z 773.055,A -85,B 0,C 180,E1 -24109.537,E2 -24109.537} C_VEL
LIN {X 0,Y 156.66,Z 774.277,A -85,B 0,C 180,E1 -24112.265,E2 -24112.265} C_VEL
LIN {X 0,Y 158.822,Z 775.037,A -85,B 0,C 180,E1 -24114.922,E2 -24114.922} C_VEL
LIN {X 0,Y 161.739,Z 775.323,A -85,B 0,C 180,E1 -24117.953,E2 -24117.953} C_VEL
LIN {X 0,Y 167.026,Z 774.587,A -85,B 0,C 180,E1 -24122.411,E2 -24122.411} C_VEL
LIN {X 0,Y 170.281,Z 773.532,A -85,B 0,C 180,E1 -24124.735,E2 -24124.735} C_VEL
LIN {X 0,Y 173.806,Z 772.029,A -85,B 0,C 180,E1 -24126.967,E2 -24126.967} C_VEL
LIN {X 0,Y 179.793,Z 768.705,A -85,B 0,C 180,E1 -24130.282,E2 -24130.282} C_VEL
LIN {X 0,Y 185.838,Z 764.528,A -85,B 0,C 180,E1 -24133.115,E2 -24133.115} C_VEL
LIN {X 0,Y 192.488,Z 758.893,A -85,B 0,C 180,E1 -24135.893,E2 -24135.893} C_VEL
LIN {X 0,Y 199.419,Z 751.901,A -85,B 0,C 180,E1 -24138.493,E2 -24138.493} C_VEL
LIN {X 0,Y 205.534,Z 744.706,A -85,B 0,C 180,E1 -24140.517,E2 -24140.517} C_VEL
LIN {X 0,Y 212.074,Z 735.592,A -85,B 0,C 180,E1 -24142.505,E2 -24142.505} C_VEL
LIN {X 0,Y 218.654,Z 724.615,A -85,B 0,C 180,E1 -24144.365,E2 -24144.365} C_VEL
LIN {X 0,Y 223.998,Z 713.642,A -85,B 0,C 180,E1 -24145.806,E2 -24145.806} C_VEL
LIN {X 0,Y 228.721,Z 701.272,A -85,B 0,C 180,E1 -24147.045,E2 -24147.045} C_VEL
LIN {X 0,Y 232.272,Z 689.174,A -85,B 0,C 180,E1 -24148.034,E2 -24148.034} C_VEL
LIN {X 0,Y 234.622,Z 677.982,A -85,B 0,C 180,E1 -24148.744,E2 -24148.744} C_VEL
LIN {X 0,Y 233.688,Z 678.345,A -85,B 0,C 180,E1 -24151.584,E2 -24151.584} C_VEL
LIN {X 0,Y 233.276,Z 679.985,A -85,B 0,C 180,E1 -24153.305,E2 -24153.305} C_VEL
LIN {X 0,Y 233.045,Z 684.963,A -85,B 0,C 180,E1 -24156.221,E2 -24156.221} C_VEL
LIN {X 0,Y 232.979,Z 685.785,A -85,B 0,C 180,E1 -24156.464,E2 -24156.464} C_VEL
LIN {X 0,Y 230.737,Z 697.577,A -85,B 0,C 180,E1 -24157.474,E2 -24157.474} C_VEL
LIN {X 0,Y 229.189,Z 703.502,A -85,B 0,C 180,E1 -24157.843,E2 -24157.843} C_VEL
LIN {X 0,Y 226.313,Z 712.304,A -85,B 0,C 180,E1 -24158.288,E2 -24158.288} C_VEL
LIN {X 0,Y 224.117,Z 717.808,A -85,B 0,C 180,E1 -24158.424,E2 -24158.424} C_VEL
LIN {X 0,Y 219.654,Z 726.62,A -85,B 0,C 180,E1 -24158.285,E2 -24158.285} C_VEL
LIN {X 0,Y 214.666,Z 735.135,A -85,B 0,C 180,E1 -24158.227,E2 -24158.227} C_VEL
LIN {X 0,Y 211.644,Z 740.071,A -85,B 0,C 180,E1 -24158.504,E2 -24158.504} C_VEL
LIN {X 0,Y 203.853,Z 752.079,A -85,B 0,C 180,E1 -24159.911,E2 -24159.911} C_VEL
LIN {X 0,Y 196.714,Z 761.643,A -85,B 0,C 180,E1 -24161.39,E2 -24161.39} C_VEL
LIN {X 0,Y 188.51,Z 771.191,A -85,B 0,C 180,E1 -24163.369,E2 -24163.369} C_VEL
LIN {X 0,Y 179.472,Z 780.327,A -85,B 0,C 180,E1 -24165.97,E2 -24165.97} C_VEL
LIN {X 0,Y 171.165,Z 787.822,A -85,B 0,C 180,E1 -24168.935,E2 -24168.935} C_VEL
LIN {X 0,Y 167.727,Z 790.833,A -85,B 0,C 180,E1 -24170.481,E2 -24170.481} C_VEL
LIN {X 0,Y 163.741,Z 801.976,A -85,B 0,C 180,E1 -24172.683,E2 -24172.683} C_VEL
LIN {X 0,Y 159.801,Z 811.508,A -85,B 0,C 180,E1 -24175.132,E2 -24175.132} C_VEL
LIN {X 0,Y 155.817,Z 820.205,A -85,B 0,C 180,E1 -24177.999,E2 -24177.999} C_VEL
LIN {X 0,Y 152.338,Z 827.381,A -85,B 0,C 180,E1 -24181.031,E2 -24181.031} C_VEL
LIN {X 0,Y 148.742,Z 834.41,A -85,B 0,C 180,E1 -24184.837,E2 -24184.837} C_VEL
LIN {X 0,Y 145.698,Z 840.003,A -85,B 0,C 180,E1 -24188.793,E2 -24188.793} C_VEL
LIN {X 0,Y 143.323,Z 844.392,A -85,B 0,C 180,E1 -24192.892,E2 -24192.892} C_VEL
LIN {X 0,Y 142.254,Z 846.71,A -85,B 0,C 180,E1 -24195.701,E2 -24195.701} C_VEL
LIN {X 0,Y 141.433,Z 848.598,A -85,B 0,C 180,E1 -24198.538,E2 -24198.538} C_VEL
LIN {X 0,Y 140.89,Z 850.021,A -85,B 0,C 180,E1 -24201.396,E2 -24201.396} C_VEL
LIN {X 0,Y 140.636,Z 851.029,A -85,B 0,C 180,E1 -24204.266,E2 -24204.266} C_VEL
LIN {X 0,Y 140.634,Z 851.766,A -85,B 0,C 180,E1 -24208.138,E2 -24208.138} C_VEL
LIN {X 0,Y 140.738,Z 851.865,A -85,B 0,C 180,E1 -24210.002,E2 -24210.002} C_VEL
LIN {X 0,Y 140.624,Z 851.631,A -85,B 0,C 180,E1 -24212.867,E2 -24212.867} C_VEL
LIN {X 0,Y 140.637,Z 851.002,A -85,B 0,C 180,E1 -24215.738,E2 -24215.738} C_VEL
LIN {X 0,Y 140.891,Z 849.983,A -85,B 0,C 180,E1 -24218.609,E2 -24218.609} C_VEL
LIN {X 0,Y 141.433,Z 848.539,A -85,B 0,C 180,E1 -24221.467,E2 -24221.467} C_VEL
LIN {X 0,Y 142.733,Z 845.55,A -85,B 0,C 180,E1 -24225.715,E2 -24225.715} C_VEL
LIN {X 0,Y 144.8,Z 841.506,A -85,B 0,C 180,E1 -24229.864,E2 -24229.864} C_VEL
LIN {X 0,Y 148.128,Z 835.275,A -85,B 0,C 180,E1 -24234.531,E2 -24234.531} C_VEL
LIN {X 0,Y 151.468,Z 828.864,A -85,B 0,C 180,E1 -24238.165,E2 -24238.165} C_VEL
LIN {X 0,Y 155.026,Z 821.547,A -85,B 0,C 180,E1 -24241.424,E2 -24241.424} C_VEL
LIN {X 0,Y 158.938,Z 813.18,A -85,B 0,C 180,E1 -24244.32,E2 -24244.32} C_VEL
LIN {X 0,Y 163.263,Z 802.825,A -85,B 0,C 180,E1 -24247.063,E2 -24247.063} C_VEL
LIN {X 0,Y 167.5,Z 791.173,A -85,B 0,C 180,E1 -24249.393,E2 -24249.393} C_VEL
LIN {X 0,Y 170.912,Z 779.435,A -85,B 0,C 180,E1 -24251.144,E2 -24251.144} C_VEL
LIN {X 0,Y 173.796,Z 767.289,A -85,B 0,C 180,E1 -24252.441,E2 -24252.441} C_VEL
LIN {X 0,Y 176.089,Z 754.408,A -85,B 0,C 180,E1 -24253.358,E2 -24253.358} C_VEL
LIN {X 0,Y 177.391,Z 740.024,A -85,B 0,C 180,E1 -24254.013,E2 -24254.013} C_VEL
LIN {X 0,Y 180.106,Z 696.144,A -85,B 0,C 180,E1 -24255.576,E2 -24255.576} C_VEL
LIN {X 0,Y 179.219,Z 674.453,A -85,B 0,C 180,E1 -24257.097,E2 -24257.097} C_VEL
LIN {X 0,Y 177.432,Z 649.78,A -85,B 0,C 180,E1 -24259.188,E2 -24259.188} C_VEL
LIN {X 0,Y 177.062,Z 646.872,A -85,B 0,C 180,E1 -24259.503,E2 -24259.503} C_VEL
LIN {X 0,Y 172.401,Z 633.713,A -85,B 0,C 180,E1 -24262.211,E2 -24262.211} C_VEL
LIN {X 0,Y 171.598,Z 631.938,A -85,B 0,C 180,E1 -24262.762,E2 -24262.762} C_VEL
LIN {X 0,Y 167.981,Z 624.251,A -85,B 0,C 180,E1 -24266.802,E2 -24266.802} C_VEL
LIN {X 0,Y 165.863,Z 619.815,A -85,B 0,C 180,E1 -24269.438,E2 -24269.438} C_VEL
LIN {X 0,Y 164.744,Z 618.173,A -85,B 0,C 180,E1 -24270.732,E2 -24270.732} C_VEL
LIN {X 0,Y 163.145,Z 614.747,A -85,B 0,C 180,E1 -24273.107,E2 -24273.107} C_VEL
LIN {X 0,Y 160.744,Z 610.665,A -85,B 0,C 180,E1 -24276.828,E2 -24276.828} C_VEL
LIN {X 0,Y 159.41,Z 608.15,A -85,B 0,C 180,E1 -24279.347,E2 -24279.347} C_VEL
LIN {X 0,Y 157.134,Z 604.379,A -85,B 0,C 180,E1 -24284.434,E2 -24284.434} C_VEL
LIN {X 0,Y 156.208,Z 602.933,A -85,B 0,C 180,E1 -24287,E2 -24287} C_VEL
LIN {X 0,Y 154.902,Z 601.081,A -85,B 0,C 180,E1 -24292.177,E2 -24292.177} C_VEL
LIN {X 0,Y 154.659,Z 599.92,A -85,B 0,C 180,E1 -24298.701,E2 -24298.701} C_VEL
LIN {X 0,Y 154.643,Z 600.127,A -85,B 0,C 180,E1 -24301.008,E2 -24301.008} C_VEL
LIN {X 0,Y 155.148,Z 601.819,A -85,B 0,C 180,E1 -24307.811,E2 -24307.811} C_VEL
LIN {X 0,Y 155.677,Z 602.871,A -85,B 0,C 180,E1 -24310.404,E2 -24310.404} C_VEL
LIN {X 0,Y 156.987,Z 606.2,A -85,B 0,C 180,E1 -24315.582,E2 -24315.582} C_VEL
LIN {X 0,Y 158.934,Z 610.583,A -85,B 0,C 180,E1 -24320.717,E2 -24320.717} C_VEL
LIN {X 0,Y 160.543,Z 614.584,A -85,B 0,C 180,E1 -24324.575,E2 -24324.575} C_VEL
LIN {X 0,Y 162.358,Z 619.415,A -85,B 0,C 180,E1 -24328.435,E2 -24328.435} C_VEL
LIN {X 0,Y 164.961,Z 627.384,A -85,B 0,C 180,E1 -24333.632,E2 -24333.632} C_VEL
LIN {X 0,Y 165.61,Z 629.08,A -85,B 0,C 180,E1 -24334.494,E2 -24334.494} C_VEL
LIN {X 0,Y 170.031,Z 636.734,A -85,B 0,C 180,E1 -24337.142,E2 -24337.142} C_VEL
LIN {X 0,Y 175.248,Z 646.711,A -85,B 0,C 180,E1 -24339.976,E2 -24339.976} C_VEL
LIN {X 0,Y 180.223,Z 658.199,A -85,B 0,C 180,E1 -24342.504,E2 -24342.504} C_VEL
LIN {X 0,Y 180.628,Z 659.836,A -85,B 0,C 180,E1 -24342.739,E2 -24342.739} C_VEL
LIN {X 0,Y 181.938,Z 675.247,A -85,B 0,C 180,E1 -24344.053,E2 -24344.053} C_VEL
LIN {X 0,Y 177.5,Z 741.222,A -85,B 0,C 180,E1 -24346.377,E2 -24346.377} C_VEL
LIN {X 0,Y 175.749,Z 754.272,A -85,B 0,C 180,E1 -24347.169,E2 -24347.169} C_VEL
LIN {X 0,Y 173.302,Z 766.915,A -85,B 0,C 180,E1 -24348.388,E2 -24348.388} C_VEL
LIN {X 0,Y 170.375,Z 778.219,A -85,B 0,C 180,E1 -24349.867,E2 -24349.867} C_VEL
LIN {X 0,Y 167.079,Z 788.593,A -85,B 0,C 180,E1 -24351.65,E2 -24351.65} C_VEL
LIN {X 0,Y 163.086,Z 799.217,A -85,B 0,C 180,E1 -24354.043,E2 -24354.043} C_VEL
